// TwinCAT 3 PLC project CNC_Base_program
// ProgramVersion: 3.1.4020.1
// libraries:
//   Tc2_CncHli, * (Beckhoff Automation GmbH)
//   Tc2_ControllerToolbox, * (Beckhoff Automation GmbH)
//   Tc2_Drive, * (Beckhoff Automation GmbH)
//   Tc2_NcDrive, * (Beckhoff Automation GmbH)
//   Tc2_NCI, * (Beckhoff Automation GmbH)
//   Tc2_PlcInterpolation, * (Beckhoff Automation GmbH)
//   Tc2_Standard, * (Beckhoff Automation GmbH)
//   Tc2_System, * (Beckhoff Automation GmbH)
//   Tc2_Utilities, * (Beckhoff Automation GmbH)
//   Tc3_Module, * (Beckhoff Automation GmbH)
// project tree:
//   DUTs/Cnc_Data_Types/HMI/ ST_HmiAxis.TcDUT, ST_HmiChannel.TcDUT, ST_HmiData.TcDUT
//   DUTs/Cnc_Data_Types/ ST_BlockSearch.TcDUT, ST_CncChannel.TcDUT, ST_CncSystem.TcDUT, ST_PosVector.TcDUT, ST_MachineMode.TcDUT, ST_ManualModeParam.TcDUT, ST_OpModes.TcDUT, ST_OpStates.TcDUT, ST_SyntaxCheck.TcDUT
//   DUTs/Cnc_Data_Types/ToolManagement/ ST_ToolData.TcDUT, ST_ToolLife.TcDUT, ST_ToolManagement.TcDUT
//   DUTs/Recipe/ RecipeHeader_Struct.TcDUT, RecipeList_Struct.TcDUT
//   DUTs/VE_VarData/ ST_VEVariableConfig.TcDUT
//   / GlobalTextList.TcGTLO, PlcTask.TcTTO, Visualization Manager.TcVMO (not stored)
//   GVLs/ Global_Manual.TcGVL, Global_Variables.TcGVL, GVL.TcGVL, IOs.TcGVL, Machining_Data.TcGVL
//   POUs/ CncAxisEnable.TcPOU, CncHFunctions.TcPOU, CncPlcManualFunctions.TcPOU, CncPlcMessages.TcPOU, CncVariables.TcPOU, CncMFunctions.TcPOU, CncRefPosOffs.TcPOU, CncPlcProgram.TcPOU, MAIN.TcPOU
//   POUs/CNC/F1_Init/ CncToolControl.TcPOU, HLI_Init.TcPOU, HLI_AxisSetControlToPlc.TcPOU, HLI_ChannelSetControlToPlc.TcPOU, HLI_UserInitialisation.TcPOU
//   POUs/CNC/F2_Operation Mode/ HLI_AxisManualMode.TcPOU, HLI_AxisReset.TcPOU, HLI_ChannelModeAuto.TcPOU, HLI_ChannelModeManual.TcPOU, HLI_ChannelModeMDI.TcPOU, HLI_ChannelModeReference.TcPOU, HLI_ChannelModeStandby.TcPOU, HLI_ChannelReset.TcPOU, MM_TEst.TcPOU, HLI_CncChannel.TcPOU
//   POUs/CNC/F3_Control/ HLI_ChannelGetActiveFeed.TcPOU, HLI_ChannelGetStatusInfo.TcPOU, HLI_ChannelResetRequest.TcPOU, HLI_ChannelSetBackwardMotion.TcPOU, HLI_ChannelSetFeedHold.TcPOU, HLI_ChannelSetHandWheelIncs.TcPOU, HLI_ChannelSetOptionalM01Stop.TcPOU, HLI_ChannelSetProgramBlockIgnore.TcPOU, HLI_ChannelSetReducedFeed.TcPOU, HLI_ChannelSetSingleBlock.TcPOU, HLI_ChannelSetSuspendAxisOutput.TcPOU, HLI_ChannelSetSyntaxCheck.TcPOU, HLI_ChannelGetError.TcPOU, HLI_ChannelGetMessage.TcPOU, HLI_ChannelGetMode.TcPOU, HLI_ChannelGetState.TcPOU, HLI_AxisSetFeedHold.TcPOU, HLI_AxisSetReferenceCam.TcPOU, HLI_AxisSetTrackingOperation.TcPOU, HLI_ChannelSetOverride.TcPOU
//   POUs/CNC/F4_MHT-Function/ HLI_ChannelResetMFunctions.TcPOU, HLI_DoChannelHFunction.TcPOU, HLI_DoChannelMFunction.TcPOU, HLI_DoChannelTFunction.TcPOU, HLI_QuitAxisMFunction.TcPOU, HLI_QuitChannelMHTFunction.TcPOU
//   POUs/CNC/F5_Variables/ LinkVEChannelStructure.TcPOU
//   POUs/CNC/F6 BlockSearch/ FB_BlockSearchRead.TcPOU, FB_BlockSearchWrite.TcPOU, HLI_ChannelBlockSearch.TcPOU
//   POUs/CNC/F9_Misc/ ADSLOG.TcPOU, ADSLOG2.TcPOU, MySystemTime.TcPOU
//   POUs/CNC/F9_Misc/HandWheel/ FB_HandWheelEnc.TcPOU, PRG_ManualModeG201.TcPOU
//   POUs/CNC/F9_Misc/Security/ CheckCNCAlive.TcPOU, SetPlcAlive.TcPOU
//   POUs/General/ DemoTest.TcPOU, DemoUpDown.TcPOU, Examples.TcPOU, FB_Flash.TcPOU, FB_AdsRead.TcPOU, FB_ReadPParamValue.TcPOU, DemoSine.TcPOU, WritePersistentData.TcPOU
//   POUs/HMI/ CncHmiData.TcPOU, DIntToString.TcPOU, FB_ReadChannelData.TcPOU, LRealToString.TcPOU, FB_ReadTechnoTFunc.TcPOU, FB_ReadTechnoMFunc.TcPOU, FB_ReadTechnoGFunc.TcPOU, FB_ReadWriteFileData.TcPOU, SetHMIVariables.TcPOU
//   POUs/Messages/ FB_SimpleEventLog.TcPOU, ShowMessages.TcPOU
//   POUs/Temperature Controller/ PCamara.TcPOU, PCamara_Out.TcPOU, PExt.TcPOU, PExt_Out.TcPOU, PTab.TcPOU, PTab_Out.TcPOU, TController_Enable.TcPOU
// real-time tasks:
//   TASK PlcTask: cycle T#10ms, priority 20, ADS port 350
//   TASK VISU_TASK: cycle T#200000us, priority 30, ADS port 351
// motion (NC):
//   TASK NC-Task 1 SAF: cycle T#2ms, priority 4, ADS port 501
//   TASK NC-Task 1 SVB: cycle T#10ms, priority 9, ADS port 511
// I/O:
//   DEVICE Device 3 (EtherCAT), AmsNetId 192.168.200.135.4.1
//     Term 1 (EK1100) [EK1100 EtherCAT Coupler (2A E-Bus)]
//       Term 2 (EL1008) [EL1008 8Ch. Dig. Input 24V, 3ms]
//       Term 3 (EL1008) [EL1008 8Ch. Dig. Input 24V, 3ms]
//       Term 4 (EL2008) [EL2008 8Ch. Dig. Output 24V, 0.5A]
//       Term 5 (EL2008) [EL2008 8Ch. Dig. Output 24V, 0.5A]
//       Term 6 (EL4024) [EL4024 4Ch. Ana. Output 4-20mA, 12bit]
//       Term 7 (EL3318) [EL3318 8Ch. Ana Input Thermocouple (TC)]
//       Term 8 (EL7037) [EL7037 1Ch. Stepper motor output stage (24V, 1.5A)] // Motor AS1020
//       Term 9 (EL7037) [EL7037 1Ch. Stepper motor output stage (24V, 1.5A)]
//       Term 10 (EL7037) [EL7037 1Ch. Stepper motor output stage (24V, 1.5A)]
//       Term 11 (EL7037) [EL7037 1Ch. Stepper motor output stage (24V, 1.5A)]
//       Term 12 (EL7037) [EL7037 1Ch. Stepper motor output stage (24V, 1.5A)]
//       Term 13 (EL7037) [EL7037 1Ch. Stepper motor output stage (24V, 1.5A)]
//       Term 14 (EL7037) [EL7037 1Ch. Stepper motor output stage (24V, 1.5A)]
//       Term 15 (EL2522) [EL2522 2Ch. Pulse Train Output]
//       Term 32 (EL7037) [EL7037 1Ch. Stepper motor output stage (24V, 1.5A)]
//       Term 16 (EL9011) [EL9011 End Terminal]
// variable links:
//   CNC/Axes/B <-> Device 3 (EtherCAT)/Term 1 (EK1100)/Term 10 (EL7037)
//     Inputs/Enc_Counter <-> ENC Status compact/Counter value
//     Inputs/Enc_Latch <-> ENC Status compact/Latch value
//     Inputs/Enc_Status @bit 4 <-> ENC Status compact/Status/Counter overflow
//     Inputs/Enc_Status @bit 3 <-> ENC Status compact/Status/Counter underflow
//     Inputs/Enc_Status @bit 7 <-> ENC Status compact/Status/Extrapolation stall
//     Inputs/Enc_Status <-> ENC Status compact/Status/Latch C valid
//     Inputs/Enc_Status @bit 1 <-> ENC Status compact/Status/Latch extern valid
//     Inputs/Enc_Status @bit 2 <-> ENC Status compact/Status/Set counter done
//     Inputs/Enc_Status2 @bit 4 <-> ENC Status compact/Status/Status of extern latch
//     Inputs/Enc_Status2 <-> ENC Status compact/Status/Status of input A
//     Inputs/Enc_Status2 @bit 1 <-> ENC Status compact/Status/Status of input B
//     Inputs/Enc_Status2 @bit 2 <-> ENC Status compact/Status/Status of input C
//     Inputs/Enc_Status2 @bit 5 <-> ENC Status compact/Status/Sync error
//     Inputs/Enc_Status2 @bit 7 <-> ENC Status compact/Status/TxPDO Toggle
//     Inputs/STM_Status @bit 11 <-> STM Status/Status/Digital input 1
//     Inputs/STM_Status @bit 12 <-> STM Status/Status/Digital input 2
//     Inputs/STM_Status @bit 3 <-> STM Status/Status/Error
//     Inputs/STM_Status @bit 7 <-> STM Status/Status/Motor stall
//     Inputs/STM_Status @bit 5 <-> STM Status/Status/Moving negative
//     Inputs/STM_Status @bit 4 <-> STM Status/Status/Moving positive
//     Inputs/STM_Status @bit 1 <-> STM Status/Status/Ready
//     Inputs/STM_Status <-> STM Status/Status/Ready to enable
//     Inputs/STM_Status @bit 13 <-> STM Status/Status/Sync error
//     Inputs/STM_Status @bit 6 <-> STM Status/Status/Torque reduced
//     Inputs/STM_Status @bit 15 <-> STM Status/Status/TxPDO Toggle
//     Inputs/STM_Status @bit 2 <-> STM Status/Status/Warning
//     Outputs/Drv_Data_Out <-> STM Velocity/Velocity
//     Outputs/Enc_Ctrl <-> ENC Control compact/Control/Enable latch C
//     Outputs/Enc_Ctrl @bit 3 <-> ENC Control compact/Control/Enable latch extern on negative edge
//     Outputs/Enc_Ctrl @bit 1 <-> ENC Control compact/Control/Enable latch extern on positive edge
//     Outputs/Enc_Ctrl @bit 2 <-> ENC Control compact/Control/Set counter
//     Outputs/STM_Ctrl <-> STM Control/Control/Enable
//     Outputs/STM_Ctrl @bit 2 <-> STM Control/Control/Reduce torque
//     Outputs/STM_Ctrl @bit 1 <-> STM Control/Control/Reset
//   CNC/Axes/C <-> Device 3 (EtherCAT)/Term 1 (EK1100)/Term 13 (EL7037)
//     Inputs/Enc_Counter <-> ENC Status compact/Counter value
//     Inputs/Enc_Latch <-> ENC Status compact/Latch value
//     Inputs/Enc_Status @bit 4 <-> ENC Status compact/Status/Counter overflow
//     Inputs/Enc_Status @bit 3 <-> ENC Status compact/Status/Counter underflow
//     Inputs/Enc_Status @bit 7 <-> ENC Status compact/Status/Extrapolation stall
//     Inputs/Enc_Status <-> ENC Status compact/Status/Latch C valid
//     Inputs/Enc_Status @bit 1 <-> ENC Status compact/Status/Latch extern valid
//     Inputs/Enc_Status @bit 2 <-> ENC Status compact/Status/Set counter done
//     Inputs/Enc_Status2 @bit 4 <-> ENC Status compact/Status/Status of extern latch
//     Inputs/Enc_Status2 <-> ENC Status compact/Status/Status of input A
//     Inputs/Enc_Status2 @bit 1 <-> ENC Status compact/Status/Status of input B
//     Inputs/Enc_Status2 @bit 2 <-> ENC Status compact/Status/Status of input C
//     Inputs/Enc_Status2 @bit 5 <-> ENC Status compact/Status/Sync error
//     Inputs/Enc_Status2 @bit 7 <-> ENC Status compact/Status/TxPDO Toggle
//     Inputs/STM_Status @bit 11 <-> STM Status/Status/Digital input 1
//     Inputs/STM_Status @bit 12 <-> STM Status/Status/Digital input 2
//     Inputs/STM_Status @bit 3 <-> STM Status/Status/Error
//     Inputs/STM_Status @bit 7 <-> STM Status/Status/Motor stall
//     Inputs/STM_Status @bit 5 <-> STM Status/Status/Moving negative
//     Inputs/STM_Status @bit 4 <-> STM Status/Status/Moving positive
//     Inputs/STM_Status @bit 1 <-> STM Status/Status/Ready
//     Inputs/STM_Status <-> STM Status/Status/Ready to enable
//     Inputs/STM_Status @bit 13 <-> STM Status/Status/Sync error
//     Inputs/STM_Status @bit 6 <-> STM Status/Status/Torque reduced
//     Inputs/STM_Status @bit 15 <-> STM Status/Status/TxPDO Toggle
//     Inputs/STM_Status @bit 2 <-> STM Status/Status/Warning
//     Outputs/Drv_Data_Out <-> STM Velocity/Velocity
//     Outputs/Enc_Ctrl <-> ENC Control compact/Control/Enable latch C
//     Outputs/Enc_Ctrl @bit 3 <-> ENC Control compact/Control/Enable latch extern on negative edge
//     Outputs/Enc_Ctrl @bit 1 <-> ENC Control compact/Control/Enable latch extern on positive edge
//     Outputs/Enc_Ctrl @bit 2 <-> ENC Control compact/Control/Set counter
//     Outputs/STM_Ctrl <-> STM Control/Control/Enable
//     Outputs/STM_Ctrl @bit 2 <-> STM Control/Control/Reduce torque
//     Outputs/STM_Ctrl @bit 1 <-> STM Control/Control/Reset
//   CNC/Axes/Extruder <-> Device 3 (EtherCAT)/Term 1 (EK1100)/Term 32 (EL7037)
//     Inputs/Enc_Counter <-> ENC Status compact/Counter value
//     Inputs/Enc_Latch <-> ENC Status compact/Latch value
//     Inputs/Enc_Status @bit 4 <-> ENC Status compact/Status/Counter overflow
//     Inputs/Enc_Status @bit 3 <-> ENC Status compact/Status/Counter underflow
//     Inputs/Enc_Status @bit 7 <-> ENC Status compact/Status/Extrapolation stall
//     Inputs/Enc_Status <-> ENC Status compact/Status/Latch C valid
//     Inputs/Enc_Status @bit 1 <-> ENC Status compact/Status/Latch extern valid
//     Inputs/Enc_Status @bit 2 <-> ENC Status compact/Status/Set counter done
//     Inputs/Enc_Status2 @bit 4 <-> ENC Status compact/Status/Status of extern latch
//     Inputs/Enc_Status2 <-> ENC Status compact/Status/Status of input A
//     Inputs/Enc_Status2 @bit 1 <-> ENC Status compact/Status/Status of input B
//     Inputs/Enc_Status2 @bit 2 <-> ENC Status compact/Status/Status of input C
//     Inputs/Enc_Status2 @bit 5 <-> ENC Status compact/Status/Sync error
//     Inputs/Enc_Status2 @bit 7 <-> ENC Status compact/Status/TxPDO Toggle
//     Inputs/STM_Status @bit 11 <-> STM Status/Status/Digital input 1
//     Inputs/STM_Status @bit 12 <-> STM Status/Status/Digital input 2
//     Inputs/STM_Status @bit 3 <-> STM Status/Status/Error
//     Inputs/STM_Status @bit 7 <-> STM Status/Status/Motor stall
//     Inputs/STM_Status @bit 5 <-> STM Status/Status/Moving negative
//     Inputs/STM_Status @bit 4 <-> STM Status/Status/Moving positive
//     Inputs/STM_Status @bit 1 <-> STM Status/Status/Ready
//     Inputs/STM_Status <-> STM Status/Status/Ready to enable
//     Inputs/STM_Status @bit 13 <-> STM Status/Status/Sync error
//     Inputs/STM_Status @bit 6 <-> STM Status/Status/Torque reduced
//     Inputs/STM_Status @bit 15 <-> STM Status/Status/TxPDO Toggle
//     Inputs/STM_Status @bit 2 <-> STM Status/Status/Warning
//     Outputs/Drv_Data_Out <-> STM Velocity/Velocity
//     Outputs/Enc_Ctrl <-> ENC Control compact/Control/Enable latch C
//     Outputs/Enc_Ctrl @bit 3 <-> ENC Control compact/Control/Enable latch extern on negative edge
//     Outputs/Enc_Ctrl @bit 1 <-> ENC Control compact/Control/Enable latch extern on positive edge
//     Outputs/Enc_Ctrl @bit 2 <-> ENC Control compact/Control/Set counter
//     Outputs/STM_Ctrl <-> STM Control/Control/Enable
//     Outputs/STM_Ctrl @bit 2 <-> STM Control/Control/Reduce torque
//     Outputs/STM_Ctrl @bit 1 <-> STM Control/Control/Reset
//   CNC/Axes/X1 <-> Device 3 (EtherCAT)/Term 1 (EK1100)/Term 8 (EL7037)
//     Inputs/Enc_Counter <-> ENC Status compact/Counter value
//     Inputs/Enc_Latch <-> ENC Status compact/Latch value
//     Inputs/Enc_Status @bit 4 <-> ENC Status compact/Status/Counter overflow
//     Inputs/Enc_Status @bit 3 <-> ENC Status compact/Status/Counter underflow
//     Inputs/Enc_Status @bit 7 <-> ENC Status compact/Status/Extrapolation stall
//     Inputs/Enc_Status <-> ENC Status compact/Status/Latch C valid
//     Inputs/Enc_Status @bit 1 <-> ENC Status compact/Status/Latch extern valid
//     Inputs/Enc_Status @bit 2 <-> ENC Status compact/Status/Set counter done
//     Inputs/Enc_Status2 @bit 4 <-> ENC Status compact/Status/Status of extern latch
//     Inputs/Enc_Status2 <-> ENC Status compact/Status/Status of input A
//     Inputs/Enc_Status2 @bit 1 <-> ENC Status compact/Status/Status of input B
//     Inputs/Enc_Status2 @bit 2 <-> ENC Status compact/Status/Status of input C
//     Inputs/Enc_Status2 @bit 5 <-> ENC Status compact/Status/Sync error
//     Inputs/Enc_Status2 @bit 7 <-> ENC Status compact/Status/TxPDO Toggle
//     Inputs/STM_Status @bit 11 <-> STM Status/Status/Digital input 1
//     Inputs/STM_Status @bit 12 <-> STM Status/Status/Digital input 2
//     Inputs/STM_Status @bit 3 <-> STM Status/Status/Error
//     Inputs/STM_Status @bit 7 <-> STM Status/Status/Motor stall
//     Inputs/STM_Status @bit 5 <-> STM Status/Status/Moving negative
//     Inputs/STM_Status @bit 4 <-> STM Status/Status/Moving positive
//     Inputs/STM_Status @bit 1 <-> STM Status/Status/Ready
//     Inputs/STM_Status <-> STM Status/Status/Ready to enable
//     Inputs/STM_Status @bit 13 <-> STM Status/Status/Sync error
//     Inputs/STM_Status @bit 6 <-> STM Status/Status/Torque reduced
//     Inputs/STM_Status @bit 15 <-> STM Status/Status/TxPDO Toggle
//     Inputs/STM_Status @bit 2 <-> STM Status/Status/Warning
//     Outputs/Drv_Data_Out <-> STM Velocity/Velocity
//     Outputs/Enc_Ctrl <-> ENC Control compact/Control/Enable latch C
//     Outputs/Enc_Ctrl @bit 3 <-> ENC Control compact/Control/Enable latch extern on negative edge
//     Outputs/Enc_Ctrl @bit 1 <-> ENC Control compact/Control/Enable latch extern on positive edge
//     Outputs/Enc_Ctrl @bit 2 <-> ENC Control compact/Control/Set counter
//     Outputs/STM_Ctrl <-> STM Control/Control/Enable
//     Outputs/STM_Ctrl @bit 2 <-> STM Control/Control/Reduce torque
//     Outputs/STM_Ctrl @bit 1 <-> STM Control/Control/Reset
//   CNC/Axes/X2 <-> Device 3 (EtherCAT)/Term 1 (EK1100)/Term 9 (EL7037)
//     Inputs/Enc_Counter <-> ENC Status compact/Counter value
//     Inputs/Enc_Latch <-> ENC Status compact/Latch value
//     Inputs/Enc_Status @bit 4 <-> ENC Status compact/Status/Counter overflow
//     Inputs/Enc_Status @bit 3 <-> ENC Status compact/Status/Counter underflow
//     Inputs/Enc_Status @bit 7 <-> ENC Status compact/Status/Extrapolation stall
//     Inputs/Enc_Status <-> ENC Status compact/Status/Latch C valid
//     Inputs/Enc_Status @bit 1 <-> ENC Status compact/Status/Latch extern valid
//     Inputs/Enc_Status @bit 2 <-> ENC Status compact/Status/Set counter done
//     Inputs/Enc_Status2 @bit 4 <-> ENC Status compact/Status/Status of extern latch
//     Inputs/Enc_Status2 <-> ENC Status compact/Status/Status of input A
//     Inputs/Enc_Status2 @bit 1 <-> ENC Status compact/Status/Status of input B
//     Inputs/Enc_Status2 @bit 2 <-> ENC Status compact/Status/Status of input C
//     Inputs/Enc_Status2 @bit 5 <-> ENC Status compact/Status/Sync error
//     Inputs/Enc_Status2 @bit 7 <-> ENC Status compact/Status/TxPDO Toggle
//     Inputs/STM_Status @bit 11 <-> STM Status/Status/Digital input 1
//     Inputs/STM_Status @bit 12 <-> STM Status/Status/Digital input 2
//     Inputs/STM_Status @bit 3 <-> STM Status/Status/Error
//     Inputs/STM_Status @bit 7 <-> STM Status/Status/Motor stall
//     Inputs/STM_Status @bit 5 <-> STM Status/Status/Moving negative
//     Inputs/STM_Status @bit 4 <-> STM Status/Status/Moving positive
//     Inputs/STM_Status @bit 1 <-> STM Status/Status/Ready
//     Inputs/STM_Status <-> STM Status/Status/Ready to enable
//     Inputs/STM_Status @bit 13 <-> STM Status/Status/Sync error
//     Inputs/STM_Status @bit 6 <-> STM Status/Status/Torque reduced
//     Inputs/STM_Status @bit 15 <-> STM Status/Status/TxPDO Toggle
//     Inputs/STM_Status @bit 2 <-> STM Status/Status/Warning
//     Outputs/Drv_Data_Out <-> STM Velocity/Velocity
//     Outputs/Enc_Ctrl <-> ENC Control compact/Control/Enable latch C
//     Outputs/Enc_Ctrl @bit 3 <-> ENC Control compact/Control/Enable latch extern on negative edge
//     Outputs/Enc_Ctrl @bit 1 <-> ENC Control compact/Control/Enable latch extern on positive edge
//     Outputs/Enc_Ctrl @bit 2 <-> ENC Control compact/Control/Set counter
//     Outputs/STM_Ctrl <-> STM Control/Control/Enable
//     Outputs/STM_Ctrl @bit 2 <-> STM Control/Control/Reduce torque
//     Outputs/STM_Ctrl @bit 1 <-> STM Control/Control/Reset
//   CNC/Axes/Y <-> Device 3 (EtherCAT)/Term 1 (EK1100)/Term 14 (EL7037)
//     Inputs/Enc_Counter <-> ENC Status compact/Counter value
//     Inputs/Enc_Latch <-> ENC Status compact/Latch value
//     Inputs/Enc_Status @bit 4 <-> ENC Status compact/Status/Counter overflow
//     Inputs/Enc_Status @bit 3 <-> ENC Status compact/Status/Counter underflow
//     Inputs/Enc_Status @bit 7 <-> ENC Status compact/Status/Extrapolation stall
//     Inputs/Enc_Status <-> ENC Status compact/Status/Latch C valid
//     Inputs/Enc_Status @bit 1 <-> ENC Status compact/Status/Latch extern valid
//     Inputs/Enc_Status @bit 2 <-> ENC Status compact/Status/Set counter done
//     Inputs/Enc_Status2 @bit 4 <-> ENC Status compact/Status/Status of extern latch
//     Inputs/Enc_Status2 <-> ENC Status compact/Status/Status of input A
//     Inputs/Enc_Status2 @bit 1 <-> ENC Status compact/Status/Status of input B
//     Inputs/Enc_Status2 @bit 2 <-> ENC Status compact/Status/Status of input C
//     Inputs/Enc_Status2 @bit 5 <-> ENC Status compact/Status/Sync error
//     Inputs/Enc_Status2 @bit 7 <-> ENC Status compact/Status/TxPDO Toggle
//     Inputs/STM_Status @bit 11 <-> STM Status/Status/Digital input 1
//     Inputs/STM_Status @bit 12 <-> STM Status/Status/Digital input 2
//     Inputs/STM_Status @bit 3 <-> STM Status/Status/Error
//     Inputs/STM_Status @bit 7 <-> STM Status/Status/Motor stall
//     Inputs/STM_Status @bit 5 <-> STM Status/Status/Moving negative
//     Inputs/STM_Status @bit 4 <-> STM Status/Status/Moving positive
//     Inputs/STM_Status @bit 1 <-> STM Status/Status/Ready
//     Inputs/STM_Status <-> STM Status/Status/Ready to enable
//     Inputs/STM_Status @bit 13 <-> STM Status/Status/Sync error
//     Inputs/STM_Status @bit 6 <-> STM Status/Status/Torque reduced
//     Inputs/STM_Status @bit 15 <-> STM Status/Status/TxPDO Toggle
//     Inputs/STM_Status @bit 2 <-> STM Status/Status/Warning
//     Outputs/Drv_Data_Out <-> STM Velocity/Velocity
//     Outputs/Enc_Ctrl <-> ENC Control compact/Control/Enable latch C
//     Outputs/Enc_Ctrl @bit 3 <-> ENC Control compact/Control/Enable latch extern on negative edge
//     Outputs/Enc_Ctrl @bit 1 <-> ENC Control compact/Control/Enable latch extern on positive edge
//     Outputs/Enc_Ctrl @bit 2 <-> ENC Control compact/Control/Set counter
//     Outputs/STM_Ctrl <-> STM Control/Control/Enable
//     Outputs/STM_Ctrl @bit 2 <-> STM Control/Control/Reduce torque
//     Outputs/STM_Ctrl @bit 1 <-> STM Control/Control/Reset
//   CNC/Axes/Z1 <-> Device 3 (EtherCAT)/Term 1 (EK1100)/Term 11 (EL7037)
//     Inputs/Enc_Counter <-> ENC Status compact/Counter value
//     Inputs/Enc_Latch <-> ENC Status compact/Latch value
//     Inputs/Enc_Status @bit 4 <-> ENC Status compact/Status/Counter overflow
//     Inputs/Enc_Status @bit 3 <-> ENC Status compact/Status/Counter underflow
//     Inputs/Enc_Status @bit 7 <-> ENC Status compact/Status/Extrapolation stall
//     Inputs/Enc_Status <-> ENC Status compact/Status/Latch C valid
//     Inputs/Enc_Status @bit 1 <-> ENC Status compact/Status/Latch extern valid
//     Inputs/Enc_Status @bit 2 <-> ENC Status compact/Status/Set counter done
//     Inputs/Enc_Status2 @bit 4 <-> ENC Status compact/Status/Status of extern latch
//     Inputs/Enc_Status2 <-> ENC Status compact/Status/Status of input A
//     Inputs/Enc_Status2 @bit 1 <-> ENC Status compact/Status/Status of input B
//     Inputs/Enc_Status2 @bit 2 <-> ENC Status compact/Status/Status of input C
//     Inputs/Enc_Status2 @bit 5 <-> ENC Status compact/Status/Sync error
//     Inputs/Enc_Status2 @bit 7 <-> ENC Status compact/Status/TxPDO Toggle
//     Inputs/STM_Status @bit 11 <-> STM Status/Status/Digital input 1
//     Inputs/STM_Status @bit 12 <-> STM Status/Status/Digital input 2
//     Inputs/STM_Status @bit 3 <-> STM Status/Status/Error
//     Inputs/STM_Status @bit 7 <-> STM Status/Status/Motor stall
//     Inputs/STM_Status @bit 5 <-> STM Status/Status/Moving negative
//     Inputs/STM_Status @bit 4 <-> STM Status/Status/Moving positive
//     Inputs/STM_Status @bit 1 <-> STM Status/Status/Ready
//     Inputs/STM_Status <-> STM Status/Status/Ready to enable
//     Inputs/STM_Status @bit 13 <-> STM Status/Status/Sync error
//     Inputs/STM_Status @bit 6 <-> STM Status/Status/Torque reduced
//     Inputs/STM_Status @bit 15 <-> STM Status/Status/TxPDO Toggle
//     Inputs/STM_Status @bit 2 <-> STM Status/Status/Warning
//     Outputs/Drv_Data_Out <-> STM Velocity/Velocity
//     Outputs/Enc_Ctrl <-> ENC Control compact/Control/Enable latch C
//     Outputs/Enc_Ctrl @bit 3 <-> ENC Control compact/Control/Enable latch extern on negative edge
//     Outputs/Enc_Ctrl @bit 1 <-> ENC Control compact/Control/Enable latch extern on positive edge
//     Outputs/Enc_Ctrl @bit 2 <-> ENC Control compact/Control/Set counter
//     Outputs/STM_Ctrl <-> STM Control/Control/Enable
//     Outputs/STM_Ctrl @bit 2 <-> STM Control/Control/Reduce torque
//     Outputs/STM_Ctrl @bit 1 <-> STM Control/Control/Reset
//   CNC/Axes/Z2 <-> Device 3 (EtherCAT)/Term 1 (EK1100)/Term 12 (EL7037)
//     Inputs/Enc_Counter <-> ENC Status compact/Counter value
//     Inputs/Enc_Latch <-> ENC Status compact/Latch value
//     Inputs/Enc_Status @bit 4 <-> ENC Status compact/Status/Counter overflow
//     Inputs/Enc_Status @bit 3 <-> ENC Status compact/Status/Counter underflow
//     Inputs/Enc_Status @bit 7 <-> ENC Status compact/Status/Extrapolation stall
//     Inputs/Enc_Status <-> ENC Status compact/Status/Latch C valid
//     Inputs/Enc_Status @bit 1 <-> ENC Status compact/Status/Latch extern valid
//     Inputs/Enc_Status @bit 2 <-> ENC Status compact/Status/Set counter done
//     Inputs/Enc_Status2 @bit 4 <-> ENC Status compact/Status/Status of extern latch
//     Inputs/Enc_Status2 <-> ENC Status compact/Status/Status of input A
//     Inputs/Enc_Status2 @bit 1 <-> ENC Status compact/Status/Status of input B
//     Inputs/Enc_Status2 @bit 2 <-> ENC Status compact/Status/Status of input C
//     Inputs/Enc_Status2 @bit 5 <-> ENC Status compact/Status/Sync error
//     Inputs/Enc_Status2 @bit 7 <-> ENC Status compact/Status/TxPDO Toggle
//     Inputs/STM_Status @bit 11 <-> STM Status/Status/Digital input 1
//     Inputs/STM_Status @bit 12 <-> STM Status/Status/Digital input 2
//     Inputs/STM_Status @bit 3 <-> STM Status/Status/Error
//     Inputs/STM_Status @bit 7 <-> STM Status/Status/Motor stall
//     Inputs/STM_Status @bit 5 <-> STM Status/Status/Moving negative
//     Inputs/STM_Status @bit 4 <-> STM Status/Status/Moving positive
//     Inputs/STM_Status @bit 1 <-> STM Status/Status/Ready
//     Inputs/STM_Status <-> STM Status/Status/Ready to enable
//     Inputs/STM_Status @bit 13 <-> STM Status/Status/Sync error
//     Inputs/STM_Status @bit 6 <-> STM Status/Status/Torque reduced
//     Inputs/STM_Status @bit 15 <-> STM Status/Status/TxPDO Toggle
//     Inputs/STM_Status @bit 2 <-> STM Status/Status/Warning
//     Outputs/Drv_Data_Out <-> STM Velocity/Velocity
//     Outputs/Enc_Ctrl <-> ENC Control compact/Control/Enable latch C
//     Outputs/Enc_Ctrl @bit 3 <-> ENC Control compact/Control/Enable latch extern on negative edge
//     Outputs/Enc_Ctrl @bit 1 <-> ENC Control compact/Control/Enable latch extern on positive edge
//     Outputs/Enc_Ctrl @bit 2 <-> ENC Control compact/Control/Set counter
//     Outputs/STM_Ctrl <-> STM Control/Control/Enable
//     Outputs/STM_Ctrl @bit 2 <-> STM Control/Control/Reduce torque
//     Outputs/STM_Ctrl @bit 1 <-> STM Control/Control/Reset
//   TC3_IEC_CNC_Sample/TC3_IEC_CNC_Sample Instance <-> Device 3 (EtherCAT)/Term 1 (EK1100)/Term 2 (EL1008)
//     PlcTask Inputs/IOs.IO_In_B <-> Channel 3/Input
//     PlcTask Inputs/IOs.IO_In_Capaci <-> Channel 7/Input
//     PlcTask Inputs/IOs.IO_In_X1 <-> Channel 1/Input
//     PlcTask Inputs/IOs.IO_In_X2 <-> Channel 2/Input
//     PlcTask Inputs/IOs.IO_In_Y <-> Channel 6/Input
//     PlcTask Inputs/IOs.IO_In_Z1 <-> Channel 4/Input
//     PlcTask Inputs/IOs.IO_In_Z2 <-> Channel 5/Input
//   TC3_IEC_CNC_Sample/TC3_IEC_CNC_Sample Instance <-> Device 3 (EtherCAT)/Term 1 (EK1100)/Term 3 (EL1008)
//     PlcTask Inputs/IOs.IO_In_Emergencia <-> Channel 8/Input
//   TC3_IEC_CNC_Sample/TC3_IEC_CNC_Sample Instance <-> Device 3 (EtherCAT)/Term 1 (EK1100)/Term 4 (EL2008)
//     PlcTask Outputs/IOs.IO_Out_Aque_Extrusor <-> Channel 7/Output
//     PlcTask Outputs/IOs.IO_Out_Aque_Mesa <-> Channel 8/Output
//     PlcTask Outputs/IOs.IO_Out_HMI <-> Channel 4/Output
//     PlcTask Outputs/IOs.IO_Out_Vent_Camara <-> Channel 6/Output
//     PlcTask Outputs/IOs.IO_Out_Vent_Porta <-> Channel 5/Output
//     PlcTask Outputs/IOs.IO_Out_Vent_Quadro1 <-> Channel 2/Output
//     PlcTask Outputs/IOs.IO_Out_Vent_Quadro2 <-> Channel 3/Output
//     PlcTask Outputs/IOs.IO_Out_Vent_cabl_X <-> Channel 1/Output
//   TC3_IEC_CNC_Sample/TC3_IEC_CNC_Sample Instance <-> Device 3 (EtherCAT)/Term 1 (EK1100)/Term 5 (EL2008)
//     PlcTask Outputs/IOs.IO_Out_Chiller <-> Channel 1/Output
//   TC3_IEC_CNC_Sample/TC3_IEC_CNC_Sample Instance <-> Device 3 (EtherCAT)/Term 1 (EK1100)/Term 6 (EL4024)
//     PlcTask Outputs/IOs.A_Out_Aque_Ar <-> AO Outputs Channel 1/Analog output
//   TC3_IEC_CNC_Sample/TC3_IEC_CNC_Sample Instance <-> Device 3 (EtherCAT)/Term 1 (EK1100)/Term 7 (EL3318)
//     PlcTask Inputs/IOs.Temp_8 <-> TC Channel 8/Value
//     PlcTask Inputs/IOs.Temp_8_status[1] <-> TC Channel 8/Status/Underrange
//     PlcTask Inputs/IOs.Temp_8_status[2] <-> TC Channel 8/Status/Overrange
//     PlcTask Inputs/IOs.Temp_8_status[3] <-> TC Channel 8/Status/Error
//     PlcTask Inputs/IOs.Temp_8_status[4] <-> TC Channel 8/Status/TxPDO State
//     PlcTask Inputs/IOs.Temp_8_status[5] <-> TC Channel 8/Status/TxPDO Toggle
//     PlcTask Inputs/IOs.Temp_Cabos <-> TC Channel 7/Value
//     PlcTask Inputs/IOs.Temp_Cabos_status[1] <-> TC Channel 7/Status/Underrange
//     PlcTask Inputs/IOs.Temp_Cabos_status[2] <-> TC Channel 7/Status/Overrange
//     PlcTask Inputs/IOs.Temp_Cabos_status[3] <-> TC Channel 7/Status/Error
//     PlcTask Inputs/IOs.Temp_Cabos_status[4] <-> TC Channel 7/Status/TxPDO State
//     PlcTask Inputs/IOs.Temp_Cabos_status[5] <-> TC Channel 7/Status/TxPDO Toggle
//     PlcTask Inputs/IOs.Temp_Camara_in <-> TC Channel 1/Value
//     PlcTask Inputs/IOs.Temp_Camara_in_status[1] <-> TC Channel 1/Status/Underrange
//     PlcTask Inputs/IOs.Temp_Camara_in_status[2] <-> TC Channel 1/Status/Overrange
//     PlcTask Inputs/IOs.Temp_Camara_in_status[3] <-> TC Channel 1/Status/Error
//     PlcTask Inputs/IOs.Temp_Camara_in_status[4] <-> TC Channel 1/Status/TxPDO State
//     PlcTask Inputs/IOs.Temp_Camara_in_status[5] <-> TC Channel 1/Status/TxPDO Toggle
//     PlcTask Inputs/IOs.Temp_Camara_out <-> TC Channel 2/Value
//     PlcTask Inputs/IOs.Temp_Camara_out_status[1] <-> TC Channel 2/Status/Underrange
//     PlcTask Inputs/IOs.Temp_Camara_out_status[2] <-> TC Channel 2/Status/Overrange
//     PlcTask Inputs/IOs.Temp_Camara_out_status[3] <-> TC Channel 2/Status/Error
//     PlcTask Inputs/IOs.Temp_Camara_out_status[4] <-> TC Channel 2/Status/TxPDO State
//     PlcTask Inputs/IOs.Temp_Camara_out_status[5] <-> TC Channel 2/Status/TxPDO Toggle
//     PlcTask Inputs/IOs.Temp_Chiller <-> TC Channel 5/Value
//     PlcTask Inputs/IOs.Temp_Chiller_status[1] <-> TC Channel 5/Status/Underrange
//     PlcTask Inputs/IOs.Temp_Chiller_status[2] <-> TC Channel 5/Status/Overrange
//     PlcTask Inputs/IOs.Temp_Chiller_status[3] <-> TC Channel 5/Status/Error
//     PlcTask Inputs/IOs.Temp_Chiller_status[4] <-> TC Channel 5/Status/TxPDO State
//     PlcTask Inputs/IOs.Temp_Chiller_status[5] <-> TC Channel 5/Status/TxPDO Toggle
//     PlcTask Inputs/IOs.Temp_Extrusor_1 <-> TC Channel 4/Value
//     PlcTask Inputs/IOs.Temp_Extrusor_1_status[1] <-> TC Channel 4/Status/Underrange
//     PlcTask Inputs/IOs.Temp_Extrusor_1_status[2] <-> TC Channel 4/Status/Overrange
//     PlcTask Inputs/IOs.Temp_Extrusor_1_status[3] <-> TC Channel 4/Status/Error
//     PlcTask Inputs/IOs.Temp_Extrusor_1_status[4] <-> TC Channel 4/Status/TxPDO State
//     PlcTask Inputs/IOs.Temp_Extrusor_1_status[5] <-> TC Channel 4/Status/TxPDO Toggle
//     PlcTask Inputs/IOs.Temp_Quadro <-> TC Channel 6/Value
//     PlcTask Inputs/IOs.Temp_Quadro_status[1] <-> TC Channel 6/Status/Underrange
//     PlcTask Inputs/IOs.Temp_Quadro_status[2] <-> TC Channel 6/Status/Overrange
//     PlcTask Inputs/IOs.Temp_Quadro_status[3] <-> TC Channel 6/Status/Error
//     PlcTask Inputs/IOs.Temp_Quadro_status[4] <-> TC Channel 6/Status/TxPDO State
//     PlcTask Inputs/IOs.Temp_Quadro_status[5] <-> TC Channel 6/Status/TxPDO Toggle
//     PlcTask Inputs/IOs.Temp_Tabuleiro <-> TC Channel 3/Value
//     PlcTask Inputs/IOs.Temp_Tabuleiro_status[1] <-> TC Channel 3/Status/Underrange
//     PlcTask Inputs/IOs.Temp_Tabuleiro_status[2] <-> TC Channel 3/Status/Overrange
//     PlcTask Inputs/IOs.Temp_Tabuleiro_status[3] <-> TC Channel 3/Status/Error
//     PlcTask Inputs/IOs.Temp_Tabuleiro_status[4] <-> TC Channel 3/Status/TxPDO State
//     PlcTask Inputs/IOs.Temp_Tabuleiro_status[5] <-> TC Channel 3/Status/TxPDO Toggle

CONFIGURATION CNC_Base_program
    RESOURCE PLC ON TwinCAT3
        TASK PlcTask(INTERVAL := T#10ms, PRIORITY := 20);
        PROGRAM MAIN WITH PlcTask : MAIN;
    END_RESOURCE
END_CONFIGURATION

// ---- DUTs/Cnc_Data_Types/HMI/ST_HmiAxis.TcDUT
TYPE ST_HmiAxis :
STRUCT
	Name								: STRING;
	actCmdPosition					: LREAL;							(* mm *)
	actVelo							: LREAL;							(* mm/min *)
	actAcc							: LREAL;							(*  *)
	// ----------------------------
	current_position_acs			: LREAL;							(* mm *)
	active_position_acs			: LREAL;							(* mm *)
	end_position_acs				: LREAL;							(* mm *)
	distanceToGo					: LREAL;							(* mm *)
END_STRUCT
END_TYPE

// ---- DUTs/Cnc_Data_Types/HMI/ST_HmiChannel.TcDUT
TYPE ST_HmiChannel :
STRUCT
   SetModeAutomatic				: BOOL;
   SetModeManual					: BOOL;
   SetModeMDI						: BOOL;
	// ----------------------------
   SetStart							: BOOL;
   SetStop							: BOOL;
   SetReset							: BOOL;
	// ----------------------------
   State								: STRING;
   Mode								: STRING;
	CommandFeed						: LREAL;
	ActiveFeed						: LREAL;
	OverrideFeedrate				: LREAL;
	NcFileName						: STRING(255);
	NcFileOffset					: DINT;
	// ----------------------------
   Error								: BOOL;
   ErrorVis							: STRING;
	ActiveProgramBuffer			: ARRAY[0..2000] OF BYTE;
	// ----------------------------
	ActiveGFuncString				: STRING;
	ActiveMFuncString				: STRING;
	ActiveTFuncString				: STRING;
	// ----------------------------
	AxisMax							: INT;
	Axis								: ARRAY[0..5] OF ST_HmiAxis;
END_STRUCT
END_TYPE

// ---- DUTs/Cnc_Data_Types/HMI/ST_HmiData.TcDUT
TYPE ST_HmiData :
STRUCT
	NumberOfChannels				: UDINT;
	Channel							: ARRAY[0..5] OF ST_HmiChannel;
END_STRUCT
END_TYPE

// ---- DUTs/Cnc_Data_Types/ST_BlockSearch.TcDUT
TYPE ST_BlockSearch :
STRUCT
   (* Block Search *)
	Active         : BOOL;
   bStartRead     : BOOL;        (* Edge signal *)
   bStartWrite    : BOOL;        (* Edge signal *)
   nType          : INT;         (* 0 - no block search
                                    3 - start position by block count
                                    4 - start position by block nr
                                    5 - start position BY individual mark *)
   fDistance      : LREAL;
   bAutoReturn    : BOOL;
   nDeviationMax  : UDINT;
   nBlockNumber   : DINT;
   nPass          : DINT;
   nBlockCount    : DINT;
END_STRUCT
END_TYPE

// ---- DUTs/Cnc_Data_Types/ST_CncChannel.TcDUT
TYPE ST_CncChannel :
STRUCT
	Mode					: ST_OpModes;									(* Operation Mode *)
	State					: ST_OpStates;									(* Operation States *)

	ActMode				: UDINT;											(* Selected Mode *)
	ActModeString		: STRING;										(* Selected Mode as string *)
	ActState				: UDINT;											(* Selected State *)
	ActStateString		: STRING;										(* Selected State as string *)

	ActDistance			: LREAL;											(* Block Search : Act. Distance *)
	ActBlockCount  	: DINT;											(* Block Search : Act. Block Count *)

	M						: ARRAY [0..MAX_M_FUNCTIONS] OF BOOL;	(* M-Functions *)
	
	
	_M						: ARRAY [0..MAX_M_FUNCTIONS] OF BOOL;	(* only internal, quit M-Functions *)
	M_Argument			: ARRAY [0..MAX_M_FUNCTIONS] OF DINT;	(* Additional M-Function parameter *)

	H						: ARRAY [1..MAX_M_FUNCTIONS] OF BOOL;	(* H-Functions *)
	_H						: ARRAY [1..MAX_M_FUNCTIONS] OF BOOL;	(* only internal, quit H-Functions *)
	H_Argument			: ARRAY [1..MAX_M_FUNCTIONS] OF DINT;	(* Additional H-Function parameter *)

	T						: ARRAY [1..MAX_T_FUNCTIONS] OF BOOL;	(* T-Functions *)
	
	ProcessStartTime	: DT;												(* Process start time *)
	ProcessEndTime		: DT;												(* Process end time *)
	ProcessRunning		: BOOL;											(* Indicates that the process is running *)
	Error					: BOOL;											(* Fehlerflag des Kanals *)
	ErrorId				: UDINT;											(* FehlerId des Kanals *)
	ErrorMask			: HLI_ERROR_MASKE;							(* Informs the user about the error location in the cnc file *)

	Message				: STRING(HLI_MSG_CONTENT_STRL);			(* Message from NC program to PLC *)
END_STRUCT
END_TYPE

// ---- DUTs/Cnc_Data_Types/ST_CncSystem.TcDUT
TYPE ST_CncSystem :
STRUCT
	bHLIInit			: BOOL;		(* Initialization of HLI done *)
	bUserInitDone	: BOOL;		(* Initialization of user data done *)
	bInitError		: BOOL;		(* Error init HLI-Interfaces *)
	nInitErrorId	: UDINT;		(* ErrorId during init HLI-Interfaces *)
	Channel			: ARRAY[0..HLI_SYS_CH_MAX] OF ST_CncChannel;
	Tool				: ARRAY[0..MAX_TOOLS] OF CNC_TOOL_DATA; (* for external tool configuration, see SysMan. channel, SDA Param, Externe Werkzeugverwaltung *)
END_STRUCT
END_TYPE

// ---- DUTs/Cnc_Data_Types/ST_PosVector.TcDUT
TYPE ST_PosVector :
STRUCT
	fPosX				: LREAL;
	fPosY				: LREAL;
	fPosZ				: LREAL;
END_STRUCT
END_TYPE

// ---- DUTs/Cnc_Data_Types/ST_MachineMode.TcDUT
TYPE ST_MachineMode :
STRUCT
	(*Mode				: ST_OpModes;	*)	(* Operation Mode *)
	(*State				: ST_OpStates;*)	(* Operation States *)

	(* Operation Mode *)
	Standby			: BOOL;
	Manual			: BOOL;
	MDI				: BOOL;
	Automatic		: BOOL;
	Homing			: BOOL;

	(* Operation State *)
	Start				: BOOL;
	Stop				: BOOL;
	Reset				: BOOL;
	Error				: BOOL;

	(* Special functions *)
	DoSingleBlock	: BOOL;
	SingleBlock		: BOOL;
   FeedHold			: BOOL;
	Backward			: BOOL;
	PrgBlockIgnore	: BOOL;
	M01Stop			: BOOL;
	BlockSearch		: ST_BlockSearch;
	SyntaxCheck    : ST_SyntaxCheck;

	(* Strings *)
	ProgramName		: STRING(1024);
	MDIString		: STRING(1024);
END_STRUCT
END_TYPE

// ---- DUTs/Cnc_Data_Types/ST_ManualModeParam.TcDUT
TYPE ST_ManualModeParam :
STRUCT
	(* manual mode parameter *)
	nOpMode				: UINT;			(* operation mode, 0-no, 1-handwheel, 2-tip, 3-jog *)
	nLogAxisNr			: UINT;			(* number of the logical axis *)
	nControlElement	: UINT;			(* number of the logical control element *)
	nHandwheelNr		: UINT;			(* number of handwheel 1..max)*)
	nHandwheelIncs		: DINT;			(* number of handwheel increments *)
	nHandwheelRes		: DINT;			(* resolution of the handwheel*)
	nTipSpeed			: UDINT;			(* speed tip mode *)
	nJogSpeed			: UDINT;			(* speed jog mode *)
	nJogDistance		: UDINT;			(* jog distance *)
	bKeyPos				: BOOL;			(* key press positive *)
	bKeyNeg				: BOOL;			(* key press negative *)
	bKeyRapid			: BOOL;			(* key press rapid *)
END_STRUCT
END_TYPE

// ---- DUTs/Cnc_Data_Types/ST_OpModes.TcDUT
TYPE ST_OpModes :
STRUCT
	Standby			: BOOL;
	Auto				: BOOL;
	Manual			: BOOL;
	MDI				: BOOL;
	Homing			: BOOL;
END_STRUCT
END_TYPE

// ---- DUTs/Cnc_Data_Types/ST_OpStates.TcDUT
TYPE ST_OpStates :
STRUCT
	Selected			: BOOL;
	Ready				: BOOL;
	Start				: BOOL;
	Stop				: BOOL;
	Reset				: BOOL;
END_STRUCT
END_TYPE

// ---- DUTs/Cnc_Data_Types/ST_SyntaxCheck.TcDUT
TYPE ST_SyntaxCheck :
STRUCT
   (* SyntaxCheck *)
   nType          : INT;	(* 
										0x0000 ISG_STANDARD Normal mode
										0x0001 SV Block search
										0x0002 SOLLKON Offline Simulation with output of setpoint data
										0x0802 SOLLKON Offline Simulation without output of setpoint data
										0x0004 ON_LINE Simulation online visualisation
										0x0008 SYNCHK Simulation syntax check
										0x0010 PROD_TIME Simulation production time computation
										0x0020 ONLINE_PROD_TIME Simulation online production time computation
										0x0040 MACHINE_LOCK Dry run without axis movement
										0x0080 TECHNO_FILTER Dry run TECHNO filter
										0x0100 KIN_TRAFO_OFF Overwrites automatic enabling for kinematic transformations by a characteristic parameter defined in SDA_MDS (sda_mds*.lis).
									*)

END_STRUCT
END_TYPE

// ---- DUTs/Cnc_Data_Types/ToolManagement/ST_ToolData.TcDUT
TYPE ST_ToolData :		(* Tool data for a tool *)
STRUCT
(* -----------------------------------------
	Hint:
--------------------------------------------
	Do not modify
		- size or type of this struct

	only modify
		- name and comment of the tool parameters
-------------------------------------------- *)

		Nr							: INT;				(* Number of the tool *)
		ToolType					: INT;				(* Type of the tool *)
		SisterTool				: INT;				(* Sister tool number *)
		ToolLocked				: INT;				(* Tool locked = 1, else = 0 *)
		ParamInt1				: INT;				(* Free int parameter of the tool *)
		ParamInt2				: INT;				(* Free int parameter of the tool *)
		ParamInt3				: INT;				(* Free int parameter of the tool *)
		ParamInt4				: INT;				(* Free int parameter of the tool *)

		Length					: LREAL;				(* Length of the tool *)
		Radius					: LREAL;				(* Radius of the tool *)
		DeltaLength				: LREAL;				(* Oversize length of the tool *)
		DeltaRadius				: LREAL;				(* Oversize radius of the tool *)
		ToolLifeTime			: LREAL;				(* Tool Life Time *)
		ToolLifeTimeMax		: LREAL;				(* Tool Life Time Max *)
		ToolLifeDistance		: LREAL;				(* Tool Life Distance *)
		ToolLifeDistanceMax	: LREAL;				(* Tool Life Distance Max *)
		Param1					: LREAL;				(* Free parameter of the tool *)
		Param2					: LREAL;				(* Free parameter of the tool *)
		Param3					: LREAL;				(* Free parameter of the tool *)
		Param4					: LREAL;				(* Free parameter of the tool *)
		Param5					: LREAL;				(* Free parameter of the tool *)
		Param6					: LREAL;				(* Free parameter of the tool *)
		Param7					: LREAL;				(* Free parameter of the tool *)
		Param8					: LREAL;				(* Free parameter of the tool *)
		Param9					: LREAL;				(* Free parameter of the tool *)
		Param10					: LREAL;				(* Free parameter of the tool *)
		Param11					: LREAL;				(* Free parameter of the tool *)
		Param12					: LREAL;				(* Free parameter of the tool *)
		Param13					: LREAL;				(* Free parameter of the tool *)
		Param14					: LREAL;				(* Free parameter of the tool *)
		Param15					: LREAL;				(* Free parameter of the tool *)
		Param16					: LREAL;				(* Free parameter of the tool *)
		Param17					: LREAL;				(* Free parameter of the tool *)
		Param18					: LREAL;				(* Free parameter of the tool *)
		Param19					: LREAL;				(* Free parameter of the tool *)
		Param20					: LREAL;				(* Free parameter of the tool *)
		Param21					: LREAL;				(* Free parameter of the tool *)
		Param22					: LREAL;				(* Free parameter of the tool *)
		Param23					: LREAL;				(* Free parameter of the tool *)
		Param24					: LREAL;				(* Free parameter of the tool *)
		Param25					: LREAL;				(* Free parameter of the tool *)
		Param26					: LREAL;				(* Free parameter of the tool *)
		Param27					: LREAL;				(* Free parameter of the tool *)
		Param28					: LREAL;				(* Free parameter of the tool *)
		Param29					: LREAL;				(* Free parameter of the tool *)
		Param30					: LREAL;				(* Free parameter of the tool *)
		(*Name					: STRING;*)
END_STRUCT
END_TYPE

// ---- DUTs/Cnc_Data_Types/ToolManagement/ST_ToolLife.TcDUT
TYPE ST_ToolLife :		(* Tool life data for a tool *)
STRUCT
	tool_id			: DINT;		(* Id of the tool *)
	res				: DINT;
	time_used		: LREAL;		(* Time of used tool in seconds *)
	dist_used		: LREAL;		(* Distance of used tool in mm *)
END_STRUCT
END_TYPE

// ---- DUTs/Cnc_Data_Types/ToolManagement/ST_ToolManagement.TcDUT
TYPE ST_ToolManagement :		(* Tool management *)
STRUCT
		ToolLife					: ST_ToolLife;		(* tool life data, PLC -> HMI *)
		ToolDataActive			: BOOL;				(* tool data activation, HMI -> PLC *)
		ToolData					: ARRAY[1..MAX_TOOLS] OF ST_ToolData;		(* tool data, HMI -> PLC *)
END_STRUCT
END_TYPE

// ---- DUTs/Recipe/RecipeHeader_Struct.TcDUT
{attribute 'pack_mode':='1'}
TYPE RecipeHeader_Struct :
STRUCT
   Name1        : STRING[40];
   Name2        : STRING[40];
   Reserve      : ARRAY[3..10] OF STRING[40];
   Values       : ARRAY[1..30] OF LREAL;
   List         : ARRAY[1..50] OF RecipeList_Struct;
END_STRUCT
END_TYPE

// ---- DUTs/Recipe/RecipeList_Struct.TcDUT
{attribute 'pack_mode':='1'}
TYPE RecipeList_Struct :
STRUCT
   ToolId       : LREAL;
   PosX         : LREAL;
   PosY         : LREAL;
   PosZ         : LREAL;
   Tool1        : LREAL;
   Tool2        : LREAL;
   Tool3        : LREAL;
   GlueTime     : LREAL;
   Velo         : LREAL;
   Reserve      : ARRAY[10..20] OF LREAL;
END_STRUCT
END_TYPE

// ---- DUTs/VE_VarData/ST_VEVariableConfig.TcDUT
TYPE ST_VEVariableConfig :
STRUCT
	VARIABLE_1		: POINTER TO ARRAY[0..3] OF DINT;
	VARIABLE_2		: POINTER TO DINT;
	VARIABLE_3		: POINTER TO BOOL;
	VARIABLE_4		: POINTER TO DINT;
	VARIABLE_5		: POINTER TO DINT;
END_STRUCT
END_TYPE

// ---- GVLs/Global_Manual.TcGVL
VAR_GLOBAL
	(***********************************
	 * Declaration for 
	 * Manual functions
	 ************************************)
	PortalInfo				: STRING;
	PortalOn					: ARRAY[1..20] OF BOOL;
	PortalOff				: ARRAY[1..20] OF BOOL;
	PortalStatus			: ARRAY[1..20] OF BYTE;

	PortalSetValueLeft	: ARRAY[1..20] OF STRING;
	PortalActValueLeft	: ARRAY[1..20] OF STRING;
	PortalSetValueRight	: ARRAY[1..20] OF STRING;
	PortalActValueRight	: ARRAY[1..20] OF STRING;

	SchweissenInfo			: STRING;
	SchweissenOn			: ARRAY[1..20] OF BOOL;
	SchweissenOff			: ARRAY[1..20] OF BOOL;
	SchweissenStatus		: ARRAY[1..20] OF BYTE;

	WerkzeugInfo			: STRING;
	WerkzeugOn				: ARRAY[1..20] OF BOOL;
	WerkzeugOff				: ARRAY[1..20] OF BOOL;
	WerkzeugStatus			: ARRAY[1..20] OF BYTE;
	

END_VAR

// ---- GVLs/Global_Variables.TcGVL
VAR_GLOBAL CONSTANT
	FIRST_MESSAGE						: INT := 1;
	LAST_MESSAGE						: INT := 50;
	
	AXIS_MANUAL_KEYUNIT_MAX			: INT := 0;		(* [0..HLI_KEY_MAXIDX(11)], 0=1 KeyUnit, 1=2 KeyUnit, ... *)	
END_VAR

VAR_GLOBAL
	CncSystem							: ST_CncSystem;
	Axis1CurrPosition: LREAL;
	Axis2CurrPosition: LREAL;
	Axis3CurrPosition: LREAL;
END_VAR

// MK check
VAR_GLOBAL
	(*--------------------------*)
	(*	Connection variables     *)
	(*--------------------------*)

	(* General signals, only for starting BDE *)
	PlcMachineMode						: ARRAY[0..5] OF ST_MachineMode;	(* HMI -> PLC *)
	PLCSelectedChannel				: INT;			(* HMI -> PLC *)

	PlcFeedOverride					: UINT;			(* HMI -> PLC *)
	PlcFeedOverride2					: UINT;			(* HMI -> PLC *)
	PlcSpindleOverride				: UINT;			(* HMI -> PLC *)

	(* PLC control signals *)
	PlcAxisEnable						: BOOL;			(* HMI -> PLC *)
	PlcDeleteFailure					: BOOL;			(* HMI -> PLC *)

	PlcReset								: BOOL;
	PlcVarWriteSettings				: BOOL;


	PlcArrayInt							: ARRAY[0..20] OF INT;
	PlcArrayReal						: ARRAY[0..10] OF REAL;
	PlcArrayString3					: ARRAY[0..10] OF STRING(50);
	PlcArrayString						: ARRAY[0..10] OF STRING;

	(* Function keys 5, 6 and 7 on the right side *)
	PlcFKeyRight5						: BOOL;
	PlcFKeyRight6						: BOOL;
	PlcFKeyRight7						: BOOL;
	
	(*--------------------------*)
	(*	BDE, PLC -> HMI          *)
	(*--------------------------*)
	BDEControlOn						: BOOL;
	BDEAutomatic						: BOOL;
	BDEVarBoolTimer					: ARRAY[0..10] OF BOOL;
	BDEVarBoolCounter					: ARRAY[0..10] OF BOOL;
	BDEVarBoolMessage					: ARRAY[0..50] OF BOOL;
	
	(* Manual Mode *)
	PlcManualModeLeftKey				: BOOL;
	PlcManualModeRightKey			: BOOL;
	PlcManualModeRapidFeedKey		: BOOL;
	PlcManualModeSelectedAxis		: UINT;
	PlcManualModeSpeed				: UDINT;
	PlcManualModeIncrements			: UDINT;
	PlcManualModeOpMode				: UINT;	(* 1-handwheel, 2-continuous, 3-Incremental, ... *)
	PlcManualModeHandWheelIncs		: DINT;
	PlcManualModeHandWheelRes		: DINT := 1;

	(*--------------------------*)
	(* Tool management          *)
	(*--------------------------*)
	PlcToolManagement					: ST_ToolManagement;
	
   (*--------------------------*)
   (* Recipe HMI -> PLC        *)
   (*--------------------------*)
   RecipeData							: RecipeHeader_Struct;
	
END_VAR

VAR_GLOBAL
	(*--------------------------*)
	(*	Messages                 *)
	(*--------------------------*)
	MSGList1								: ARRAY [FIRST_MESSAGE..LAST_MESSAGE] OF BOOL;
	MSGListQuit1						: ARRAY [FIRST_MESSAGE..LAST_MESSAGE] OF BOOL;
	MSGList2								: ARRAY [FIRST_MESSAGE..LAST_MESSAGE] OF BOOL;
	MSGListQuit2						: ARRAY [FIRST_MESSAGE..LAST_MESSAGE] OF BOOL;
	MSGList3								: ARRAY [FIRST_MESSAGE..LAST_MESSAGE] OF BOOL;
	MSGListQuit3						: ARRAY [FIRST_MESSAGE..LAST_MESSAGE] OF BOOL;
	MSGList4								: ARRAY [FIRST_MESSAGE..LAST_MESSAGE] OF BOOL;
	MSGListQuit4						: ARRAY [FIRST_MESSAGE..LAST_MESSAGE] OF BOOL;
END_VAR

VAR_GLOBAL PERSISTENT
	test1									: INT;
	test2									: INT;
	test3									: INT;
END_VAR

VAR_GLOBAL
	(*--------------------------*)
	(*	Temperatura             *)
	(*--------------------------*)
	Temp_Camara_set			: DINT :=0;						(*0.01ºC*)
	Temp_Tabuleiro_set		: DINT :=0;						(*0.01ºC*)
	Temp_Extrusor_1_set		: DINT :=0;						(*0.1ºC*)
	Temp_Extrusor_2_set		: DINT :=0;						(*0.1ºC*)

END_VAR

// ---- GVLs/GVL.TcGVL
{attribute 'qualified_only'}
VAR_GLOBAL
	Temp_Camara_in :INT;
	Temp_Tabuleiro :INT;
	Temp_Extrusor_1 :INT;
	Temp_Chiller :INT;
	Temp_Quadro :INT;
	Temp_Cabos:INT;
	Temp_8:INT;
	Temp_MotorB:LREAL:=50.0;
	Temp_PontoMovel:LREAL:=50.0;
	gvl_bstate_start :BOOL:= FALSE;
	gvl_sprogramname :STRING(500) := '';
	gvl_currentState :DWORD;
	gvl_automaticstop :BOOL :=FALSE;
	gvl_automaticreset :BOOL :=FALSE;
	gvl_automaticselected :BOOL :=FALSE;
	gvl_bEnableTracking:BOOL:=FALSE;
	gvl_plcAxisEnable:BOOL:=FALSE;
	gvl_operationMode:STRING(100):='';
	gvl_manualMode:BOOL;
	gvl_automaticMode:BOOL;
	gvl_machine_state:STRING(500):='';
	gvl_blockcount:DINT:=0;
	gvl_aquecimento_mesa:BOOL :=FALSE;
	gvl_aquecimento_extrusor:BOOL :=FALSE;
	gvl_manualmode_isactivated:BOOL :=FALSE;
	gvl_manualmode_busy:BOOL :=FALSE;
	gvl_currentMode:DWORD;
	gvl_Manual_nOpMode:UINT;
END_VAR

// ---- GVLs/IOs.TcGVL
VAR_GLOBAL
	IO_In1				AT %I*		: BOOL;
	IO_In2				AT %I*		: BOOL;
	IO_In3				AT %I*		: BOOL;
	IO_In4				AT %I*		: BOOL;

	IO_Out1				AT %Q*		: BOOL;
	IO_Out2				AT %Q*		: BOOL;
	IO_Out3				AT %Q*		: BOOL;
	IO_Out4				AT %Q*		: BOOL;
	
	
	//Definição dos inputs/outputs cartas de I/O
	
	IO_Out_Vent_cabl_X	AT %Q*		: BOOL;
	IO_Out_Vent_Quadro1	AT %Q*		: BOOL;
	IO_Out_Vent_Quadro2	AT %Q*		: BOOL;
	IO_Out_HMI			AT %Q*		: BOOL;
	IO_Out_Vent_Porta	AT %Q*		: BOOL;
	IO_Out_Vent_Camara	AT %Q*		: BOOL;
	IO_Out_Aque_Extrusor	AT %Q*		: BOOL;
	IO_Out_Aque_Mesa	AT %Q*		: BOOL;
	IO_Out_Chiller		AT %Q*		: BOOL;
	A_Out_Aque_Ar		AT %Q*		: UINT;
	
	IO_In_X1			AT %I*		: BOOL;
	IO_In_X2			AT %I*		: BOOL;
	IO_In_B				AT %I*		: BOOL;
	IO_In_Z1			AT %I*		: BOOL;
	IO_In_Z2			AT %I*		: BOOL;
	IO_In_Y				AT %I*		: BOOL;
	IO_In_Capaci		AT %I*		: BOOL;
	IO_In_Emergencia	AT %I*		: BOOL;
	
	//Inputs Temperatura
	
	Temp_Camara_in			AT %I*			: INT;						(*0.01ºC*)
	Temp_Camara_in_status	AT %I*			: ARRAY [1..5] OF BOOL;		(*Underrange; Overrange; Error; TxPDO State; TxPDO Toggle*)
	
	Temp_Camara_out			AT %I*			: INT;						(*0.01ºC*)
	Temp_Camara_out_status	AT %I*			: ARRAY [1..5] OF BOOL;		(*Underrange; Overrange; Error; TxPDO State; TxPDO Toggle*)
	
	Temp_Tabuleiro			AT %I*			: INT;						(*0.01ºC*)
	Temp_Tabuleiro_status	AT %I*			: ARRAY [1..5] OF BOOL;		(*Underrange; Overrange; Error; TxPDO State; TxPDO Toggle*)
	
	Temp_Extrusor_1			AT %I*			: INT;						(*0.1ºC*)
	Temp_Extrusor_1_status	AT %I*			: ARRAY [1..5] OF BOOL;		(*Underrange; Overrange; Error; TxPDO State; TxPDO Toggle*)
	
	Temp_Chiller			AT %I*			: INT;						(*0.1ºC*)
	Temp_Chiller_status		AT %I*			: ARRAY [1..5] OF BOOL;		(*Underrange; Overrange; Error; TxPDO State; TxPDO Toggle*)
	
	Temp_Quadro				AT %I*			: INT;						(*0.1ºC*)
	Temp_Quadro_status		AT %I*			: ARRAY [1..5] OF BOOL;		(*Underrange; Overrange; Error; TxPDO State; TxPDO Toggle*)
	
	Temp_Cabos				AT %I*			: INT;						(*0.1ºC*)
	Temp_Cabos_status		AT %I*			: ARRAY [1..5] OF BOOL;		(*Underrange; Overrange; Error; TxPDO State; TxPDO Toggle*)
	
	Temp_8					AT %I*			: INT;						(*0.1ºC*)
	Temp_8_status			AT %I*			: ARRAY [1..5] OF BOOL;		(*Underrange; Overrange; Error; TxPDO State; TxPDO Toggle*)
	
END_VAR

// ---- GVLs/Machining_Data.TcGVL
VAR_GLOBAL CONSTANT
	(* General limits *)
	MAX_TOOLS								: UINT := 50;
	SystemToolNr							: INT := 30;		(* System Tool Number *)
	
	MAX_TIMER								: INT := 50;
	MAX_M_FUNCTIONS						: UDINT := 200;
	MAX_T_FUNCTIONS						: UDINT := 200;

	(* BDE - Messages *)
	BDE_MSG_1								: INT := 1;
	BDE_MSG_2								: INT := 2;
	BDE_MSG_3								: INT := 3;

	(* BDE - Timer *)
	BDE_TIMER_SUM							: INT := 1;
	BDE_TIMER_CONTROL_ON					: INT := 2;
	BDE_TIMER_AUTOMATIC					: INT := 3;
	BDE_TIMER_ERROR						: INT := 4;

	(* BDE - Counter *)
	BDE_COUNTER_AUTO						: INT := 1;
	BDE_COUNTER_PIECES					: INT := 2;
END_VAR

VAR_GLOBAL
	(*--------------------------*)
	(*	Machine data table       *)
	(*--------------------------*)
	PLCMParBool				: ARRAY[1..10] OF BOOL;
	PLCMParInt				: ARRAY[1..50] OF INT;
	PLCMParByte				: ARRAY[1..20] OF BYTE;
	PLCMParDInt				: ARRAY[1..70] OF DINT;
	PLCMParUSInt			: ARRAY[1..20] OF USINT;
	PLCMParUInt				: ARRAY[1..20] OF UINT;
	PLCMParUDInt			: ARRAY[1..20] OF UDINT;
	PLCMParReal				: ARRAY[1..90] OF REAL;
	PLCMParLReal			: ARRAY[1..90] OF LREAL;
	PLCMParString			: ARRAY[1..50] OF STRING;
	PLCMParTime				: ARRAY[1..50] OF TIME;

	PLCMParList1			: ARRAY[1..100] OF LREAL;
	PLCMParList2			: ARRAY[1..50] OF LREAL;
	PLCMParList3			: ARRAY[1..50] OF LREAL;
	PLCMParListString		: ARRAY[1..50] OF STRING;
	PLCMParTimer			: ARRAY[1..50] OF TIME;
END_VAR

VAR_GLOBAL
	(* Timer *)
	PlcTimer					: ARRAY[1..MAX_TIMER] OF REAL;

	(* General Machining data *)
	MachineParam			: ARRAY[1..50] OF REAL;
	TestBol					: ARRAY[1..50] OF BOOL;
END_VAR

// ---- POUs/MAIN.TcPOU
PROGRAM MAIN

(* ========================================================= *)
(*    PRG: TwinCAT CNC                                       *)
(* --------------------------------------------------------- *)
(*  Desc: Base PLC program for TwinCAT CNC                  *)
(* 	Author: MK                                                *)
(*  Date: 21.12.2011                                        *)
(*  Cust.:                                                   *)
(*  M-No:                                                   *)
(*  Kom.:                                                   *)
(*  Rev.: 1.3  from 1.24                                    *)
(* ========================================================= *)

DemoSine();
DemoUpDown();
DemoTest();
WritePersistentData();
ShowMessages();
MySystemTime();

HLI_Init();
IF CncSystem.bHLIInit = TRUE THEN
	CncPlcProgram();
	CncMFunctions();
	CncPlcManualFunctions();
	CncPlcMessages();
	CncRefPosOffs();
	CncVariables();
	CncHmiData();
	
	//gpAx[0]^.ipo_mc_control.emergency_stop.command_w :=1;
	
	//Axis1CurrPosition := gpAx[0]^.lr_state.current_position_acs_r/10000.0;
	//Axis2CurrPosition := gpAx[0]^.lr_state.current_position_acs_r/10000.0;
	//Axis3CurrPosition := gpAx[0]^.lr_state.current_position_acs_r/10000.0;
	
END_IF



								(*--Belo Controlador--*)
TController_Enable();
								
								(* -- Set das variáveis para a HMI -- *)
SetHMIVariables();

END_PROGRAM

// ---- POUs/General/DemoSine.TcPOU
PROGRAM DemoSine
VAR
	X_Value		: REAL;
	Y_Value		: REAL;
	Y_ValueAbs	: REAL;

	maxValue		: INT := 1000;
	index			: INT;
END_VAR

(* ========================================================= *)
(*    PRG: DemoSine                                          *)
(* --------------------------------------------------------- *)
(*   Desc: Example, shows how to generate a sine             *)
(* Author: MK                                                *)
(*   Date: 21.12.2011                                        *)
(*   Rev.: 1.0                                               *)
(* ========================================================= *)


IF index >= maxValue THEN
	index := 0;
ELSE
	index := index + 1;
END_IF

X_Value := INT_TO_REAL(index)/INT_TO_REAL(maxValue) * 2.0 * 3.1415;
Y_Value := SIN(X_Value) * 100.0;
Y_ValueAbs := (Y_Value+100.0)/2.0;

END_PROGRAM

// ---- POUs/General/DemoUpDown.TcPOU
PROGRAM DemoUpDown
VAR
	bGo				: BOOL;
	UpDown			: INT;
END_VAR

(* ========================================================= *)
(*    PRG: DemoUpDown                                        *)
(* --------------------------------------------------------- *)
(*   Desc: Example, shows how to generate a up down signal   *)
(* Author: MK                                                *)
(*   Date: 21.12.2011                                        *)
(*   Rev.: 1.0                                               *)
(* ========================================================= *)


(* up down counter *)
IF bGo THEN
	UpDown := UpDown - 1;
	IF UpDown < 1 THEN
		bGo := FALSE;
	END_IF
ELSE
	UpDown := UpDown + 1;
	IF UpDown >= 100 THEN
		bGo := TRUE;
	END_IF
END_IF

END_PROGRAM

// ---- POUs/General/DemoTest.TcPOU

PROGRAM DemoTest
VAR_INPUT
	bEnable					: BOOL := TRUE;
END_VAR
VAR
	HandWheelEnc			: FB_HandWheelEnc;
	incs						: UDINT;
	dir						: INT;
	testTOD					: TOD;
	testDT					: DT;
	testTime					: TIME;
	testUInt32				: UDINT;
	nColor					: UDINT := 16#5522AA;
	stPosVector				: ST_PosVector;
END_VAR

IF bEnable = TRUE THEN
	PortalActValueLeft[3] := INT_TO_STRING(DemoUpDown.UpDown);
	PortalActValueLeft[4] := INT_TO_STRING(DemoUpDown.UpDown);
	PortalActValueLeft[5] := INT_TO_STRING(DemoUpDown.UpDown);
END_IF


IF dir = 0 THEN
	;
ELSIF dir = 1 THEN
	incs := incs + 1;
	
	IF incs > 1024 THEN
		incs := 0;
	END_IF
ELSIF dir = 2 THEN 
	incs := incs - 1;

	IF incs < 0 THEN
		incs := 1024;
	END_IF
END_IF

HandWheelEnc(EncoderValue:=incs);


stPosVector.fPosX := CncHmiData.PlcHmiData.Channel[0].Axis[0].active_position_acs;
stPosVector.fPosY := CncHmiData.PlcHmiData.Channel[0].Axis[1].active_position_acs;
stPosVector.fPosZ := CncHmiData.PlcHmiData.Channel[0].Axis[2].active_position_acs;

END_PROGRAM

// ---- POUs/CNC/F9_Misc/HandWheel/FB_HandWheelEnc.TcPOU
FUNCTION_BLOCK FB_HandWheelEnc
VAR_INPUT
   EncoderValue         : UDINT;
   EncoderValueMax      : DINT := 65535;		//  := 1024;
END_VAR
VAR_OUTPUT
   OUT                  : DINT;
END_VAR
VAR
   oldEncoderValue      : UDINT;
   nTurns               : DINT;
END_VAR

(* ========================================================= *)
(*     FB: FB_HandWheelEnc                                   *)
(* --------------------------------------------------------- *)
(*   Desc: Handles encoder overflow                          *)
(* Author: MK                                                *)
(*   Date: 20.10.2015                                        *)
(*   Rev.: 1.1                                               *)
(* ========================================================= *)


IF UDINT_TO_DINT(oldEncoderValue - EncoderValue) >  EncoderValueMax/2 THEN		// positiv overflow
	nTurns := nTurns + 1;
ELSIF UDINT_TO_DINT(EncoderValue - oldEncoderValue) > EncoderValueMax/2 THEN	// negativ overflow
	nTurns := nTurns - 1;
END_IF

oldEncoderValue := EncoderValue;

OUT := nTurns * EncoderValueMax + UDINT_TO_DINT(EncoderValue);

END_FUNCTION_BLOCK

// ---- POUs/HMI/CncHmiData.TcPOU
PROGRAM CncHmiData
VAR_INPUT
END_VAR
VAR
	PlcHmiData						: ST_HmiData;
	nChIdx							: UDINT;
	fbReadChannelData				: ARRAY[0..5] OF FB_ReadChannelData;
END_VAR

(* ========================================================= *)
(*    FUN: CncHmiData                                        *)
(* --------------------------------------------------------- *)
(*   Desc:                                                   *)
(* Author: MK                                                *)
(*   Date: 01.12.2015                                        *)
(*   Rev.: 1.0                                               *)
(* ========================================================= *)


//RETURN;

PlcHmiData.NumberOfChannels := gpPform^.nc_config.number_of_channels_r;
FOR nChIdx := 0 TO PlcHmiData.NumberOfChannels - 1 DO
	fbReadChannelData[nChIdx](nChIdx:=nChIdx, pHmiChannel:=ADR(PlcHmiData.Channel[nChIdx]));
END_FOR

END_PROGRAM

// ---- POUs/HMI/FB_ReadChannelData.TcPOU
FUNCTION_BLOCK FB_ReadChannelData
VAR_INPUT
	nChIdx							: UDINT;
	pHmiChannel						: POINTER TO ST_HmiChannel;
END_VAR
VAR_OUTPUT
END_VAR
VAR
	pChannel							: POINTER TO HIGH_LEVEL_INTERFACE_CH;
	pAx								: POINTER TO HIGH_LEVEL_INTERFACE_AX;

	timerFileName					: TON;
	sFileName						: STRING(255);
	sFileNameOld					: STRING(255);
	sTmp								: STRING(255);

	nFileOffset						: DINT;
	nFileOffsetOld					: DINT := -1;
	
	fbReadWriteData				: FB_ReadWriteFileData;
	bReadFileErr					: BOOL;
	bReadNcFile						: BOOL;
	bReadFileActive				: BOOL;

	timerTechno						: TON;
	bReadTechnoInfoActive		: BOOL;	
	fbReadTechnoGFunc				: FB_ReadTechnoGFunc;
	fbReadTechnoMFunc				: FB_ReadTechnoMFunc;
	fbReadTechnoTFunc				: FB_ReadTechnoTFunc;
	
	fbFlash							: FB_Flash;
	nAxIdx							: INT;
END_VAR

(* ========================================================= *)
(*    FUN: FB_ReadChannelData                                *)
(* --------------------------------------------------------- *)
(*   Desc:                                                   *)
(* Author: MK                                                *)
(*   Date: 01.12.2015                                        *)
(*   Rev.: 1.0                                               *)
(* ========================================================= *)


(* get pointer to channel data *)
pChannel := gpCh[nChIdx];
IF pChannel = 0 THEN
	RETURN;
END_IF

(* commanded feedrade *)
pHmiChannel^.CommandFeed := pChannel^.bahn_state.command_feed_r/1000.0*60.0;		(* mm/min *)

(* active feedrade *)
pHmiChannel^.ActiveFeed := pChannel^.bahn_state.active_feed_r/1000.0*60.0;			(* mm/min *)

(* override *)
pHmiChannel^.OverrideFeedrate := pChannel^.bahn_mc_control.override_feedrate.state_r/10.0;		(* % *)


(* read file name and file offset *)
timerFileName(IN := NOT(timerFileName.Q), PT := T#150MS);
IF timerFileName.Q THEN
	(*MRODRIGUES
	sFileName := pChannel^.bahn_state.file_name_r.zeichen;*)
	sFileName := GVL.gvl_sprogramname;
	nFileOffset := pChannel^.bahn_state.active_fileoffset_r;
	pHmiChannel^.NcFileName := sFileName;
	pHmiChannel^.NcFileOffset := nFileOffset;

	IF sFileNameOld <> sFileName OR nFileOffsetOld <> nFileOffset THEN
		sFileNameOld := sFileName;
		nFileOffsetOld := nFileOffset;
		bReadNcFile := TRUE;
	END_IF
END_IF

(* read nc file data *)
IF (bReadNcFile = TRUE OR bReadFileActive = TRUE) THEN
	IF sFileName = ''  
		OR LEFT(STR:=sFileName, SIZE:=3) = 'C:\'
	THEN
		sTmp := sFileName;
	ELSE
		(* sub program, add default path *)
		sTmp := CONCAT('c:\twincat\cnc\', sFileName);
	END_IF
	
	fbReadWriteData(sNetId := '',
							sPathName := sTmp,
							nSeekPos := pHmiChannel^.NcFileOffset,
							bExecute := bReadNcFile,
							bWrite := FALSE,
							pBuffer := ADR(pHmiChannel^.ActiveProgramBuffer),
							nBufferSize := SIZEOF(pHmiChannel^.ActiveProgramBuffer)-1,
							bError => bReadFileErr,
							bBusy => bReadFileActive);
	bReadNcFile := FALSE;

	IF fbReadWriteData.bBusy = FALSE AND fbReadWriteData.bError = FALSE THEN
		bReadFileErr := FALSE;
	END_IF
END_IF


(* read technology information *)
timerTechno(IN := NOT(timerTechno.Q), PT := T#500MS);
IF timerTechno.Q THEN
	bReadTechnoInfoActive := TRUE;
END_IF

IF bReadTechnoInfoActive THEN
	fbReadTechnoGFunc(nIdxGrp	:= 16#20100 + 1 + nChIdx,
							nIdxOffs	:= 16#03C,
							nLen		:= 2*40,
							bStart	:= timerTechno.Q,
							pStr		:= ADR(pHmiChannel^.ActiveGFuncString));
							
	fbReadTechnoMFunc(nIdxGrp	:= 16#20100 + 1 + nChIdx,
							nIdxOffs	:= 16#03D,
							nLen		:= 4*40,
							bStart	:= timerTechno.Q,
							pStr		:= ADR(pHmiChannel^.ActiveMFuncString));

	fbReadTechnoTFunc(nIdxGrp	:= 16#20100 + 1 + nChIdx,
							nIdxOffs	:= 16#01A,
							nLen		:= 4,
							bStart	:= timerTechno.Q,
							pStr		:= ADR(pHmiChannel^.ActiveTFuncString));
							
	IF fbReadTechnoGFunc.bBusy = FALSE
		AND fbReadTechnoMFunc.bBusy = FALSE
		AND fbReadTechnoTFunc.bBusy = FALSE
	THEN
		bReadTechnoInfoActive := FALSE;
	END_IF
END_IF


(* channel mode and state *) 
pHmiChannel^.Mode := CncSystem.Channel[nChIdx+1].ActModeString;
pHmiChannel^.State := CncSystem.Channel[nChIdx+1].ActStateString;


(* channel mode Automatic, Manual, MDI *)
IF pHmiChannel^.SetModeAutomatic = TRUE THEN
	PlcMachineMode[nChIdx+1].Automatic := pHmiChannel^.SetModeAutomatic;
	pHmiChannel^.SetModeAutomatic := FALSE;
	IF PlcMachineMode[nChIdx+1].ProgramName = '' THEN
		PlcMachineMode[nChIdx+1].ProgramName := 'c:\TwinCAT\Cnc\Stadion.nc';
	END_IF
END_IF

IF pHmiChannel^.SetModeManual = TRUE THEN
	PlcMachineMode[nChIdx+1].Manual := pHmiChannel^.SetModeManual;
	pHmiChannel^.SetModeManual := FALSE;
END_IF

IF pHmiChannel^.SetModeMDI = TRUE THEN
	PlcMachineMode[nChIdx+1].MDI := pHmiChannel^.SetModeMDI;
	pHmiChannel^.SetModeMDI := FALSE;
END_IF

(* Channel start, stop, reset *)
IF pHmiChannel^.SetStart = TRUE THEN
	PlcMachineMode[1].Start := pHmiChannel^.SetStart;
	pHmiChannel^.SetStart := FALSE;
END_IF

IF pHmiChannel^.SetStop = TRUE THEN
	PlcMachineMode[nChIdx+1].Stop := pHmiChannel^.SetStop;
	pHmiChannel^.SetStop := FALSE;
END_IF

IF pHmiChannel^.SetReset = TRUE THEN
	PlcMachineMode[nChIdx+1].Reset := pHmiChannel^.SetReset;
	pHmiChannel^.SetReset := FALSE;
END_IF


(* Channel Error *) 
fbFlash();

IF HLI_ChannelGetState(nChan := nChIdx+1) = 6 THEN
	pHmiChannel^.Error := TRUE;
	
	IF fbFlash.bFlash = TRUE THEN
		pHmiChannel^.ErrorVis := 'Visible';
	ELSE
		pHmiChannel^.ErrorVis := 'Hidden';
	END_IF
ELSE
	pHmiChannel^.Error := FALSE;
	pHmiChannel^.ErrorVis := 'Hidden';
END_IF


(* axis data *)
FOR nAxIdx := 0 TO 10 DO
	IF	pChannel^.bahn_state.coord_r[nAxIdx].log_achs_nr_r = 0 THEN
		CONTINUE;
	END_IF

	pHmiChannel^.AxisMax := nAxIdx + 1;
	pHmiChannel^.Axis[nAxIdx].Name := pChannel^.bahn_state.coord_r[naxIdx].axis_name_r.zeichen;
	
	pAx := gpAx[naxIdx];
	pHmiChannel^.Axis[nAxIdx].actCmdPosition := pAx^.ipo_state.s_act/10000.0;		(* mm *)
	pHmiChannel^.Axis[nAxIdx].actVelo := pAx^.ipo_state.v_act/1000.0*60.0;			(* mm/min *) 
	pHmiChannel^.Axis[nAxIdx].actAcc := pAx^.ipo_state.a_act/1000.0;					(*  *)
	
	pHmiChannel^.Axis[nAxIdx].current_position_acs := pAx^.lr_state.current_position_acs_r/10000.0;		(* mm *)
	pHmiChannel^.Axis[nAxIdx].active_position_acs := pAx^.lr_state.active_position_acs_r/10000.0;		(* mm *)
	pHmiChannel^.Axis[nAxIdx].end_position_acs := pAx^.lr_state.end_position_acs_r/10000.0;				(* mm *)
	pHmiChannel^.Axis[nAxIdx].distanceToGo := pHmiChannel^.Axis[nAxIdx].end_position_acs - pHmiChannel^.Axis[nAxIdx].active_position_acs;						(* mm *)
END_FOR

END_FUNCTION_BLOCK

// ---- POUs/HMI/FB_ReadWriteFileData.TcPOU
FUNCTION_BLOCK FB_ReadWriteFileData
VAR_INPUT
	sNetId						: T_AmsNetId;		(* TwinCAT network address of the file *)
	sPathName					: T_MaxString;		(* File path and name *)
	nSeekPos						: DINT;				(* New seek pointer position *)
	bExecute						: BOOL;
	bWrite						: BOOL;				(* TRUE => Write, FALSE => Read *)
	tTimeOut						: TIME := DEFAULT_ADS_TIMEOUT;	(* Max. ADS timeout time *)
	pBuffer						: POINTER TO BYTE;
	nBufferSize					: UDINT;
END_VAR
VAR_OUTPUT
	bBusy							: BOOL;				(* TRUE => execution in progress, FALSE => execution idle *)
	bError						: BOOL;
	nErrId						: UDINT;
END_VAR
VAR
   nStep							: DWORD;
	nModeTmp						: DWORD;
	RisingEdge					: R_TRIG;
	hFile							: UINT := 0;		(* file handle *)
	fbFileOpen					: FB_FileOpen;
	fbFileClose					: FB_FileClose;
	fbFileRead					: FB_FileRead;
	fbFileWrite					: FB_FileWrite;
	fbFileSeek					: FB_FileSeek;
	bStepReady					: BOOL;
END_VAR

IF sPathName = '' THEN
	IF bWrite = FALSE THEN
		pBuffer^ := 0;
	END_IF
	RisingEdge(CLK:=FALSE);
	bBusy := FALSE;
	bError := FALSE;
	nErrId := 0;
	RETURN;
END_IF


RisingEdge(CLK:=bExecute);

CASE nStep OF
	0:		(* idle *)
		IF RisingEdge.Q THEN
			bBusy := TRUE;
			bError := FALSE;
			nErrId := 0;
			hFile := 0;
			
			IF bWrite = FALSE THEN
				nModeTmp := FOPEN_MODEREAD OR FOPEN_MODEBINARY;
			ELSE
				nModeTmp := FOPEN_MODEWRITE OR FOPEN_MODEBINARY;
			END_IF

			(*--- open file ---*)
			fbFileOpen(bExecute:=FALSE);
			fbFileOpen(sNetId:=sNetId, sPathName:=sPathName,
							nMode:=nModeTmp, ePath:=PATH_GENERIC,
							tTimeout:=tTimeOut, bExecute:=TRUE);
							
			IF NOT fbFileOpen.bBusy THEN
					bError := TRUE;
				ELSE
					bError := false;
				END_IF
							
			IF nSeekPos <> 0 THEN
				nStep := 10;
			ELSE
				nStep := 11;
			END_IF
		END_IF


	10:	(*--- wait for open finished and seek ---*)
		fbFileOpen(bExecute:=FALSE);
		IF NOT fbFileOpen.bBusy THEN
			IF fbFileOpen.bError THEN
				nErrId := fbFileOpen.nErrId;
				bError := TRUE;
				nStep := 50;
			ELSE
				hFile := fbFileOpen.hFile;

				(*--- seek file pointer ---*)
				fbFileSeek(bExecute:=FALSE);
				fbFileSeek(sNetId:=sNetId, hFile:=hFile,  
								nSeekPos:=nSeekPos, eOrigin:=SEEK_SET,
								bExecute:=TRUE, tTimeout:=tTimeOut);
				nStep := 11;
			END_IF
		END_IF
		

	11:	(*--- wait for open/seek finished and read/write---*)
		bStepReady := FALSE;
		IF nSeekPos = 0 THEN
			(*--- wait for open finished ---*)
			fbFileOpen(bExecute:=FALSE);
			IF NOT fbFileOpen.bBusy THEN
				IF fbFileOpen.bError THEN
					nErrId := fbFileOpen.nErrId;
					bError := TRUE;
					nStep := 50;
				ELSE
					hFile := fbFileOpen.hFile;
					bStepReady := TRUE;
				END_IF
			END_IF
		ELSE
			(*--- wait for seek finished ---*)
			fbFileSeek(bExecute:=FALSE);
			IF NOT fbFileSeek.bBusy THEN
				IF fbFileSeek.bError THEN
					nErrId := fbFileSeek.nErrId;
					bError := TRUE;
					nStep := 50;
				ELSE
					bStepReady := TRUE;
				END_IF
			END_IF
		END_IF
		
		IF bStepReady = TRUE THEN
			IF bWrite = FALSE THEN
				(*--- read data from file ---*)
				MEMSET(pBuffer, 0, nBufferSize);
				fbFileRead(bExecute:=FALSE);
				fbFileRead(sNetId:=sNetId, hFile:=hFile,
								pReadBuff:=pBuffer, cbReadLen:=nBufferSize,
								bExecute:=TRUE, tTimeout:=tTimeOut);
				nStep := 20;
			ELSE
				(*--- write data to file ---*)
				fbFileWrite(bExecute:=FALSE);
				fbFileWrite(sNetId:=sNetId, hFile:=hFile,
								pWriteBuff:=pBuffer, cbWriteLen:=nBufferSize,
								bExecute:=TRUE, tTimeout:=tTimeOut);
				nStep := 21;
			END_IF
		END_IF


	20:	(*--- wait for read finished and close---*)
		fbFileRead(bExecute := FALSE);
		IF NOT fbFileRead.bBusy THEN
			IF fbFileRead.bError THEN
				nErrId := fbFileRead.nErrId;
				bError := TRUE;
				nStep := 50;
			ELSE
				(*--- close the file ---*)
				fbFileClose(bExecute:=FALSE);
				fbFileClose(sNetId:=sNetId, hFile:=hFile, bExecute:=TRUE, tTimeout:=tTimeOut);
				nStep := 30;
			END_IF
		END_IF


	21:	(*--- wait for write finished and close ---*)
		fbFileWrite(bExecute:=FALSE);
		IF NOT fbFileWrite.bBusy THEN
			IF fbFileWrite.bError THEN
				nErrId := fbFileWrite.nErrId;
				bError := TRUE;
				nStep := 50;
			ELSE
				(*--- close the file ---*)
				fbFileClose(bExecute:=FALSE);
				fbFileClose(sNetId:=sNetId, hFile:=hFile, bExecute:=TRUE, tTimeout:=tTimeOut);
				nStep := 30;
			END_IF
		END_IF


	30:	(*--- wait for close finished ---*)
		fbFileClose(bExecute:=FALSE);
		IF NOT fbFileClose.bBusy THEN
			IF fbFileClose.bError THEN
				nErrId := fbFileClose.nErrId;
				bError := TRUE;
				nStep := 50;
			ELSE
				hFile := 0;
				nStep := 0;			(* ready *)
				bBusy := FALSE;
			END_IF
		END_IF

	50:	(*--- Error ---*)
		IF (hFile <> 0) THEN
			(*--- try close the file ---*)
			fbFileClose(bExecute:=FALSE);
			fbFileClose(sNetId:=sNetId, hFile:=hFile, bExecute:=TRUE, tTimeout:=tTimeOut);
			nStep := 30;		(* wait for close *)
		ELSE
			nStep := 0;			(* ready *)
			bBusy := FALSE;
		END_IF

END_CASE

END_FUNCTION_BLOCK

// ---- POUs/HMI/FB_ReadTechnoGFunc.TcPOU
FUNCTION_BLOCK FB_ReadTechnoGFunc
VAR_INPUT
   sNetId               : T_AmsNetId;
   nPort                : T_AmsPort := 553;
   nIdxGrp              : UDINT;
   nIdxOffs             : UDINT;
	nLen						: UDINT;
   bStart               : BOOL;
	pStr						: POINTER TO STRING;
END_VAR
VAR_OUTPUT
   bBusy                : BOOL;
   bErr                 : BOOL;
END_VAR
VAR
   fbRead               : ADSREAD;
   bStarted             : BOOL;
   destArr               : ARRAY[0..40] OF INT;
	i							: INT;
	tmp						: STRING;
END_VAR

(* ========================================================= *)
(*     FB: FB_ReadTechnoGFunc                                *)
(* --------------------------------------------------------- *)
(*   Desc: Reads the technology information                  *)
(*       : from the CNC                                      *)
(* Author: MK                                                *)
(*   Date: 21.12.2011                                        *)
(*   Rev.: 1.0                                               *)
(* ========================================================= *)


IF bStart = TRUE AND bStarted = FALSE THEN
	bStarted := TRUE;
	bErr := FALSE;
	bBusy := TRUE;
END_IF

IF bStarted THEN
   fbRead(NetID:=sNetId, Port:=nPort, IdxGrp:=nIdxGrp, IdxOffs:=nIdxOffs,
         LEN:=nLen, DestAddr:=ADR(destArr), READ:=bStarted, TMOUT:=DEFAULT_ADS_TIMEOUT);
   IF NOT fbRead.Busy THEN
      IF fbRead.Err THEN
         bErr := TRUE;
		ELSE
			tmp := '';
			FOR i:=0 TO 36 DO
				IF destArr[i] <> -1 THEN
					tmp := CONCAT(tmp, 'G');
					tmp := CONCAT(tmp, INT_TO_STRING(destArr[i]));
					tmp := CONCAT(tmp, ' ');
		      END_IF
			END_FOR
			pStr^ := tmp;
      END_IF
      fbRead(READ := FALSE);
      bStarted := FALSE;
      bBusy := FALSE;
   END_IF
END_IF

END_FUNCTION_BLOCK

// ---- POUs/HMI/FB_ReadTechnoMFunc.TcPOU
FUNCTION_BLOCK FB_ReadTechnoMFunc
VAR_INPUT
   sNetId               : T_AmsNetId;
   nPort                : T_AmsPort := 553;
   nIdxGrp              : UDINT;
   nIdxOffs             : UDINT;
	nLen						: UDINT;
   bStart               : BOOL;
	pStr						: POINTER TO STRING;
END_VAR
VAR_OUTPUT
   bBusy                : BOOL;
   bErr                 : BOOL;
END_VAR
VAR
   fbRead               : ADSREAD;
   bStarted             : BOOL;
   destArr             : ARRAY[0..40] OF UDINT;
	i							: UDINT;
	nMax						: UDINT;
	tmp						: STRING;
END_VAR

(* ========================================================= *)
(*     FB: FB_ReadTechnoMFunc                                *)
(* --------------------------------------------------------- *)
(*   Desc: Reads the technology information                  *)
(*       : from the CNC                                      *)
(* Author: MK                                                *)
(*   Date: 21.12.2011                                        *)
(*   Rev.: 1.0                                               *)
(* ========================================================= *)


IF bStart = TRUE AND bStarted = FALSE THEN
	bStarted := TRUE;
	bErr := FALSE;
	bBusy := TRUE;
END_IF

IF bStarted THEN
   fbRead(NetID:=sNetId, Port:=nPort, IdxGrp:=nIdxGrp, IdxOffs:=nIdxOffs,
         LEN:=nLen, DestAddr:=ADR(destArr), READ:=bStarted, TMOUT:=DEFAULT_ADS_TIMEOUT);
   IF NOT fbRead.Busy THEN
      IF fbRead.Err THEN
         bErr := TRUE;
		ELSE
			tmp := '';
			nMax := destArr[0];
			FOR i:=1 TO nMax DO
				IF destArr[i] <> -1 THEN
					tmp := CONCAT(tmp, 'M');
					tmp := CONCAT(tmp, UDINT_TO_STRING(destArr[i]));
					tmp := CONCAT(tmp, ' ');
		      END_IF
			END_FOR
			pStr^ := tmp;
      END_IF
      fbRead(READ := FALSE);
      bStarted := FALSE;
      bBusy := FALSE;
   END_IF
END_IF

END_FUNCTION_BLOCK

// ---- POUs/HMI/FB_ReadTechnoTFunc.TcPOU
FUNCTION_BLOCK FB_ReadTechnoTFunc
VAR_INPUT
   sNetId               : T_AmsNetId;
   nPort                : T_AmsPort := 553;
   nIdxGrp              : UDINT;
   nIdxOffs             : UDINT;
	nLen						: UDINT;
   bStart               : BOOL;
	pStr						: POINTER TO STRING;
END_VAR
VAR_OUTPUT
   bBusy                : BOOL;
   bErr                 : BOOL;
END_VAR
VAR
   fbRead               : ADSREAD;
   bStarted             : BOOL;
   dest                 : UDINT;
	i							: INT;
	tmp						: STRING;
END_VAR

(* ========================================================= *)
(*     FB: FB_ReadTechnoTFunc                                *)
(* --------------------------------------------------------- *)
(*   Desc: Reads the technology information                  *)
(*       : from the CNC                                      *)
(* Author: MK                                                *)
(*   Date: 21.12.2011                                        *)
(*   Rev.: 1.0                                               *)
(* ========================================================= *)


IF bStart = TRUE AND bStarted = FALSE THEN
	bStarted := TRUE;
	bErr := FALSE;
	bBusy := TRUE;
END_IF

IF bStarted THEN
   fbRead(NetID:=sNetId, Port:=nPort, IdxGrp:=nIdxGrp, IdxOffs:=nIdxOffs,
         LEN:=nLen, DestAddr:=ADR(dest), READ:=bStarted, TMOUT:=DEFAULT_ADS_TIMEOUT);
   IF NOT fbRead.Busy THEN
      IF fbRead.Err THEN
         bErr := TRUE;
		ELSE
			tmp := 'T';
			tmp := CONCAT(tmp, UDINT_TO_STRING(dest));
			pStr^ := tmp;
      END_IF
      fbRead(READ := FALSE);
      bStarted := FALSE;
      bBusy := FALSE;
   END_IF
END_IF

END_FUNCTION_BLOCK

// ---- POUs/General/FB_Flash.TcPOU
FUNCTION_BLOCK FB_Flash
VAR_INPUT
	tiTime_On							: TIME := T#0.5S;		(* Zeitwert für Blinkbit ein *)
	tiTime_Off							: TIME := T#0.5s;		(* Zeitwert für Blinkbit aus *)
END_VAR
VAR_OUTPUT
	bFlash								: BOOL;					(* Blinkbit *)
END_VAR
VAR
	tnTimer_ON							: TON;
	tnTimer_OFF							: TON;
END_VAR

tnTimer_OFF(IN:=tnTimer_ON.Q, PT:=tiTime_On);
tnTimer_ON(IN:=NOT tnTimer_OFF.Q, PT:=tiTime_Off);
bFlash := tnTimer_ON.Q;

END_FUNCTION_BLOCK

// ---- POUs/CNC/F3_Control/HLI_ChannelGetState.TcPOU
FUNCTION HLI_ChannelGetState : DWORD
VAR_INPUT
	nChan					: UDINT;			(* Number of channel *)
END_VAR
VAR
	nHliChIdx			: UDINT;
END_VAR

(* ========================================================= *)
(*    FUN: HLI_ChannelGetState                               *)
(* --------------------------------------------------------- *)
(*   Desc:                                                   *)
(* Author: MK                                                *)
(*   Date: 21.12.2011                                        *)
(*   Rev.: 1.0                                               *)
(* ========================================================= *)


nHliChIdx := nChan - 1;

IF nChan <= 0 OR gNrCh < nChan OR			(* check for channel no *)
	gpCh[nHliChIdx] = 0 THEN					(* check for zero pointer *)
	HLI_ChannelGetState := 0;
	RETURN; (* e x i t *)
END_IF

(* if the stop button from the HMI is selected the request is set *)
HLI_ChannelGetState := gpCh[nHliChIdx]^.channel_mc_control.mode_and_state.state_r.state;

END_FUNCTION

// ---- POUs/General/WritePersistentData.TcPOU
PROGRAM WritePersistentData
VAR
	bWriteData							: BOOL;
	fbWritePersistentData			: FB_WritePersistentData;
	rtWriteData							: R_TRIG;
	bIsActive							: BOOL;

	Busy									: BOOL;
	ERR									: BOOL;
	ERRID									: UDINT;
	fbFlash1								: FB_Flash;
	bGo									: BOOL := false;
END_VAR


fbFlash1(tiTime_On := T#10MS, tiTime_Off := T#10MS);
bWriteData := fbFlash1.bFlash and bGo;

rtWriteData(CLK:=bWriteData);
IF rtWriteData.Q THEN
	bIsActive := TRUE;
END_IF


IF bIsActive THEN
	fbWritePersistentData(NETID:='', PORT:=851, START:=bIsActive, TMOUT:=T#1s, MODE := SPDM_2PASS);
	IF fbWritePersistentData.BUSY = FALSE THEN
		fbWritePersistentData(START:=FALSE);
		bIsActive := FALSE;
	END_IF
END_IF

Busy := fbWritePersistentData.BUSY;
ERR := fbWritePersistentData.ERR;
ERRID := fbWritePersistentData.ERRID;

END_PROGRAM

// ---- POUs/Messages/ShowMessages.TcPOU
PROGRAM ShowMessages
VAR
	SimpleEventLog1		: FB_SimpleEventLog;
	SimpleEventLog2		: FB_SimpleEventLog;
	SimpleEventLog3		: FB_SimpleEventLog;
	SimpleEventLog4		: FB_SimpleEventLog;

	bStart					: BOOL;

	bClear					: BOOL := TRUE;
	ClearEvents				: ADSCLEAREVENTS;

	bSetMsg1					: BOOL;
	bSetMsg2					: BOOL;
END_VAR

(* ----------------------------------------------------------
	Clears all active and logged events at startup.
	Should only be used at the startup sequence!
	During PLC runtime cycle each event has to be handled with
	set event, acknowledge event and or quit event!
	Don't use ClearEvents in any other case!!!
   ---------------------------------------------------------- *)
IF bClear THEN
  ClearEvents(NetID:='', bClear:=TRUE, iMode:=TCEVENTLOGIOFFS_CLEARALL, tTimeout:= t#1s);
  bClear := FALSE;
ELSE
  ClearEvents(bClear:=FALSE);
END_IF;


(* ----------------------------------------------------------
	Shows how to display messages.
	At startup the different message lists are set up.
	If new message lists are added, don't forget to restart again!

	The different message classes are listed below.

	TCEVENTCLASS_NONE				:=0,	 No class
	TCEVENTCLASS_MAINTENANCE	:=1,	 Maintenance hint
	TCEVENTCLASS_MESSAGE			:=2,	 Message
	TCEVENTCLASS_HINT				:=3,	 Hint
	TCEVENTCLASS_STATEINFO		:=4,	 State information
	TCEVENTCLASS_INSTRUCTION	:=5,	 Instruction
	TCEVENTCLASS_WARNING			:=6,	 Warning
	TCEVENTCLASS_ALARM			:=7,	 Alarm
	TCEVENTCLASS_PARAMERROR		:=8	 Parameter error
   ---------------------------------------------------------- *)

IF NOT bStart THEN
	bStart := TRUE;
	SimpleEventLog1(Init				:= TRUE,
						SourceId			:= 50,
						Class				:= TCEVENTCLASS_WARNING,
						QuitRequired	:= FALSE,
						adrAlarmArray	:= ADR(MSGList1),
						adrQuitArray	:= ADR(MSGListQuit1));

	SimpleEventLog2(Init				:= TRUE,
						SourceId			:= 51,
						Class				:= TCEVENTCLASS_ALARM,
						QuitRequired	:= FALSE,
						adrAlarmArray	:= ADR(MSGList2),
						adrQuitArray	:= ADR(MSGListQuit2));

	SimpleEventLog3(Init				:= TRUE,
						SourceId			:= 52,
						Class				:= TCEVENTCLASS_INSTRUCTION,
						QuitRequired	:= FALSE,
						adrAlarmArray	:= ADR(MSGList3),
						adrQuitArray	:= ADR(MSGListQuit3));

	SimpleEventLog4(Init				:= TRUE,
						SourceId			:= 1000,
						Class				:= TCEVENTCLASS_ALARM,
						QuitRequired	:= FALSE,
						adrAlarmArray	:= ADR(MSGList4),
						adrQuitArray	:= ADR(MSGListQuit4));
ELSE
	SimpleEventLog1(Init:=FALSE);
	SimpleEventLog2(Init:=FALSE);
	SimpleEventLog3(Init:=FALSE);
	SimpleEventLog4(Init:=FALSE);
END_IF

END_PROGRAM

// ---- POUs/Messages/FB_SimpleEventLog.TcPOU
(*****************************************************************************************
Name:				FB_SimpleEventLog
Date:				13.10.2004
Author:			Dirk Nordberg (BECKHOFF INDUSTRIE ELEKTRONIK)

Description: Function block to control the EventLogger
	Messages can be activated or deactivated through an array of bool.
	The subscription of the array is equivalent to EventID from EventLogger.
	Funtion block will be initialized with Init flag, then the busy flag is set true. 

	Revision:	1.3
	History:		13.10.2004	Ng	start coding
					17.04.2005	MK	runtime optimized
					07.07.2005	MK	short puls BF
*****************************************************************************************)
FUNCTION_BLOCK FB_SimpleEventLog
VAR_INPUT
	Init				: BOOL;				(* Rising flag starts the initialization *)
	SourceId			: UINT;				(* Number of the source Id *)
	Class				: UINT;				(* Alarm error class *)
	QuitRequired	: BOOL;				(* Activate or deaktivate confirmation *)
	adrAlarmArray	: POINTER TO BOOL;(* Adress of the array for the messages *)
												(* ...with constant boundaries ARRAY_LBOUND to ARRAY_UBOUND for array size *)
	adrQuitArray	: POINTER TO BOOL;(* Adress of the array for the confirmations	*)
												(* ...with constant boundaries ARRAY_LBOUND to ARRAY_UBOUND for array size *)
END_VAR
VAR_OUTPUT
	Busy				: BOOL;
	Err 				: BOOL;
	ErrId			 	: UDINT;
END_VAR
VAR CONSTANT
	ARRAY_LBOUND				: INT := FIRST_MESSAGE;
	ARRAY_UBOUND				: INT := LAST_MESSAGE;
	TCEVENTDATAFORMATSTRING	: STRING := ' ';
	STATE_INIT					: INT := 0;
	STATE_IDLE					: INT := 1;
	STATE_RESET_EVENT			: INT := 2;
	STATE_QUIT_EVENT			: INT := 3;
	STATE_RESET_END			: INT := 4;
	STATE_WAIT					: INT := 5;
END_VAR
VAR
	state					: INT;
(*{flag nowatch on }*)
	bReady				: BOOL := TRUE;
	nMsgHasChanged		: DINT;
	bEvtState			: ARRAY [ARRAY_LBOUND..ARRAY_UBOUND] OF BOOL;
	event					: ARRAY [ARRAY_LBOUND..ARRAY_UBOUND] OF ADSLOGEVENT;
	idx					: INT;
	CfgEvent				: TcEvent;
	bWait					: BOOL;
	ptAlarm				: POINTER TO BOOL;
	ptQuit				: POINTER TO BOOL;
	RT_Init				: R_TRIG;
(*{flag off}*)
END_VAR


nMsgHasChanged := MEMCMP(ADR(bEvtState), adrAlarmArray, SIZEOF(bEvtState));
RT_Init(CLK:=Init);

CASE State OF
	STATE_INIT:		(* Set the parameter for TcEvent *)
		Err := FALSE;
		ErrId :=0;
		Busy := FALSE;
		CfgEvent.Prio := 0;
		CfgEvent.DataFormatStrAddress := ADR(TCEVENTDATAFORMATSTRING);
		CfgEvent.Flags := TCEVENTFLAG_LOG OR TCEVENTFLAG_SRCID;
		CfgEvent.StreamType := TCEVENTSTREAM_SIMPLE;
		CfgEvent.ProgId := 'TcEventFormatter.TcXmlFormatter';
		CfgEvent.Prio := 1;
		CfgEvent.SourceId := SourceId;
		CfgEvent.Class := Class ;
		CfgEvent.bQuitRequired := QuitRequired;
		FOR idx := ARRAY_LBOUND TO ARRAY_UBOUND BY 1 DO
			CfgEvent.Id := idx;
			event[idx](NETID:='', PORT:=110, Event:=FALSE , EventQuit:=FALSE,
				 EventConfigData:=CfgEvent, FbCleanup:=FALSE, TMOUT:=t#1s);
		END_FOR;
		State := STATE_IDLE;

	STATE_IDLE:
		(* nothing to do *)
		IF nMsgHasChanged = 0
			AND bReady = TRUE
			AND NOT RT_Init.Q THEN
			RETURN;
		END_IF

		IF adrAlarmArray <> 0 THEN
			ptAlarm := adrAlarmArray;
			IF CfgEvent.bQuitRequired AND adrQuitArray <> 0 THEN
				ptQuit := adrQuitArray;
				FOR idx := ARRAY_LBOUND TO ARRAY_UBOUND BY 1 DO
					event[idx](Event:=ptAlarm^, EventQuit:=ptQuit^);
					ptAlarm := ptAlarm + 1;
					ptQuit := ptQuit + 1;
				END_FOR;
			ELSE
				bReady := TRUE;
				FOR idx := ARRAY_LBOUND TO ARRAY_UBOUND BY 1 DO
					event[idx](Event:=ptAlarm^);
					IF (NOT(ptAlarm^ = TRUE
							AND event[idx].Event = TRUE		(* event is set/on *)
							AND event[idx].Quit = FALSE
							AND event[idx].EventState = TCEVENTSTATE_SIGNALED)
						AND NOT (ptAlarm^ = FALSE
							AND event[idx].Event = FALSE		(* event is reset/off *)
							AND event[idx].Quit = TRUE
							AND event[idx].EventState = TCEVENTSTATE_INVALID)) THEN
						bReady := FALSE;
					END_IF
					ptAlarm := ptAlarm + 1;
				END_FOR;

				(* copy the status *)
				IF bReady THEN
					MEMCPY(ADR(bEvtState), adrAlarmArray, SIZEOF(bEvtState));
				END_IF

			END_IF
		END_IF

		IF RT_Init.Q THEN
			Busy := TRUE;
			State := STATE_RESET_EVENT;
		END_IF

	STATE_RESET_EVENT:(*---------------------------------- clear messages ----------------------------------------*)
		FOR idx := ARRAY_LBOUND TO ARRAY_UBOUND BY 1 DO
			IF event[idx].EventState = TCEVENTSTATE_SIGNALED THEN
				event[idx](Event:=FALSE, EventQuit:= FALSE, FbCleanup:= FALSE, TMOUT:= t#1s);
				IF event[idx].Err THEN
					Err := TRUE;
					ErrId := event[idx].ErrId;
					IF event[idx].ErrId = 1282 THEN	(* Message Router: mailbox full *)
						event[idx](Event:=FALSE, EventQuit:= FALSE, FbCleanup:= FALSE);
						RETURN;
					END_IF
				END_IF
			END_IF;
		END_FOR;
		State := STATE_QUIT_EVENT;

	STATE_QUIT_EVENT:(*---------------------------------- quit messages ----------------------------------------*)
		FOR idx := ARRAY_LBOUND TO ARRAY_UBOUND BY 1 DO
			IF event[idx].EventState = TCEVENTSTATE_SIGNALED THEN
				event[idx](Event:=FALSE, EventQuit:= TRUE, FbCleanup:= FALSE, TMOUT:= t#1s);
				IF event[idx].Err THEN
					Err := TRUE;
					ErrId := event[idx].ErrId;
					IF event[idx].ErrId = 1282 THEN	(* Message Router: mailbox full *)
						event[idx](Event:=FALSE, EventQuit:= FALSE, FbCleanup:= FALSE);
						RETURN;
					END_IF
				END_IF
			END_IF;
		END_FOR;
		State := STATE_RESET_END;

	STATE_RESET_END:
		bWait := FALSE;
		FOR idx := ARRAY_LBOUND TO ARRAY_UBOUND BY 1 DO
			event[idx](Event:=FALSE, EventQuit:= FALSE, FbCleanup:= FALSE);
			IF event[idx].EventState = TCEVENTSTATE_SIGNALED THEN
				bWait := TRUE;
			END_IF
		END_FOR;
		IF NOT bWait THEN
			State := STATE_INIT;
		END_IF

END_CASE

END_FUNCTION_BLOCK

// ---- POUs/CNC/F9_Misc/MySystemTime.TcPOU
PROGRAM MySystemTime
VAR
	nState								: INT;
	fbGetTime							: NT_GetTime;
	tonGetTime							: TON;
	bSystemTimeValid					: BOOL := FALSE;
	bFirstCycle							: BOOL;

	ptBaseTime							: TIME := t#1000ms;
	ptTime								: TIME := t#1000ms;
	dtSystemTime						: DT;
	stSystemTime						: TIMESTRUCT;
	sTime 								: STRING;		(*long date, time string*)
	sShortTime 							: STRING;		(*short time string*)
	sShortDate 							: STRING;		(*short date string*)
	nDayShortDate						: WORD;

	(* time zone information *)
	wHour									: WORD := 99;
	tzID									: E_TimeZoneID := eTimeZoneID_Invalid;
																(*	eTimeZoneID_Invalid := -1,
																	eTimeZoneID_Unknown := 0,
																	eTimeZoneID_Standard := 1,
																	eTimeZoneID_Daylight := 2 *)
	fbGetTimeZoneInformation		: FB_GetTimeZoneInformation;
END_VAR

(* Read the time *)

IF bFirstCycle = FALSE THEN
	bFirstCycle := TRUE;
	(* 970 = 1000 - 30 bei 10ms, 930 = 1000 - 60 bei 20ms ??? 921-940 *)
	ptBaseTime := T#1000MS - UDINT_TO_TIME(3 * TwinCAT_SystemInfoVarList._TaskInfo[1].CycleTime/10000);
	ptTime := ptBaseTime;
END_IF


CASE nState OF
	0:
		tonGetTime(IN := TRUE, PT := ptTime);
		IF tonGetTime.Q THEN
			tonGetTime(IN := FALSE);
			nState := 10;
		END_IF

	10:
		fbGetTime(START := TRUE);
		IF fbGetTime.BUSY = FALSE THEN
			stSystemTime := fbGetTime.TIMESTR;
			dtSystemTime := SYSTEMTIME_TO_DT(fbGetTime.TIMESTR);
			fbGetTime(START := FALSE);
			sTime := SYSTEMTIME_TO_STRING(stSystemTime);
			sShortTime := MID(STR:=sTime, LEN:=8, POS:=12);

			(* build short date string *)
			IF nDayShortDate <> MySystemTime.stSystemTime.wDay THEN
				nDayShortDate := MySystemTime.stSystemTime.wDay;
				(* day *)
				IF MySystemTime.stSystemTime.wDay < 10 THEN
					sShortDate := CONCAT(STR1:='0', STR2:=DWORD_TO_STRING(MySystemTime.stSystemTime.wDay));
				ELSE
					sShortDate := DWORD_TO_STRING(MySystemTime.stSystemTime.wDay);
				END_IF
				sShortDate := CONCAT(STR1:=sShortDate, STR2:='.');
				(* month *)
				IF MySystemTime.stSystemTime.wMonth < 10 THEN
					sShortDate := CONCAT(STR1:=sShortDate, STR2:='0');
					sShortDate := CONCAT(STR1:=sShortDate, STR2:=DWORD_TO_STRING(MySystemTime.stSystemTime.wMonth));
				ELSE
					sShortDate := CONCAT(STR1:=sShortDate, STR2:=DWORD_TO_STRING(MySystemTime.stSystemTime.wMonth));
				END_IF
				(* year *)
				sShortDate := CONCAT(STR1:=sShortDate, STR2:='.');
				sShortDate := CONCAT(STR1:=sShortDate, STR2:=DWORD_TO_STRING(MySystemTime.stSystemTime.wYear));
			END_IF

			bSystemTimeValid := TRUE;
			nState := 0;

			IF stSystemTime.wMilliseconds > 30 THEN
				ptTime := ptBaseTime - t#20ms;
			ELSIF stSystemTime.wMilliseconds < 7 THEN
				ptTime := ptBaseTime + T#20MS;
			ELSE
				ptTime := ptBaseTime;
			END_IF
		END_IF

END_CASE


(* get time zone information, summer/winter, only once a day *)
IF MySystemTime.stSystemTime.wHour <> wHour THEN
	IF MySystemTime.stSystemTime.wHour = 4 OR wHour = 99 THEN

		fbGetTimeZoneInformation(bExecute := TRUE);
		IF fbGetTimeZoneInformation.bBusy = FALSE THEN
			fbGetTimeZoneInformation(bExecute := FALSE);
			tzID := fbGetTimeZoneInformation.tzID;
			wHour := MySystemTime.stSystemTime.wHour;
		END_IF

	ELSE
		wHour := MySystemTime.stSystemTime.wHour;
	END_IF
END_IF

END_PROGRAM

// ---- POUs/CNC/F1_Init/HLI_Init.TcPOU
PROGRAM HLI_Init
VAR
	HliInterface		: MCV_HliInterface;
	tool					: CncToolControl;
	MessageOutput		: R_TRIG;
	
	bFirstCycle			: BOOL := TRUE;
	bInitHLI				: BOOL;
END_VAR

(* ========================================================= *)
(*    PRG: HLI_Init                                          *)
(* --------------------------------------------------------- *)
(*   Desc:                                                   *)
(* Author: MK                                                *)
(*   Date: 21.12.2011                                        *)
(*   Rev.: 1.0                                               *)
(* ========================================================= *)


(* Init Tool Configuration structures *)
tool.HandleExternalToolData();
tool.SetToolData();


IF NOT bInitHLI THEN
	HliInterface();
	IF HliInterface.Initialized = TRUE THEN
		bInitHLI := TRUE;
	END_IF
END_IF

IF HliInterface.Initialized = TRUE AND HliInterface.Error = FALSE THEN
	(* User initialization, used during start of PLC once *)
	IF CncSystem.bUserInitDone = FALSE THEN
		(* Initialisierungen auf dem HLI-Interface *)
		CncSystem.bUserInitDone := HLI_UserInitialisation();

		ADSLOG(strMsg:='High Level Interfaces initialized: %s', nDINT:=0, strArg:='');
	END_IF

	(* initialization finished *)
	CNCSystem.bHLIInit := TRUE;
ELSE
	MessageOutput(CLK:=HliInterface.Error);
	IF HliInterface.Error = TRUE	THEN
		(* Fehler beim Initialisieren des HLI *)
		IF MessageOutput.Q THEN
			ADSLOGDINT(	msgCtrlMask := ADSLOG_MSGTYPE_ERROR OR
												ADSLOG_MSGTYPE_MSGBOX OR
												ADSLOG_MSGTYPE_LOG,
							msgFmtStr := 'Fehler beim Initialisieren des HLI-Interfaces Fehlercode: %d',
							dintArg := HliInterface.ErrorID);
		END_IF
		CNCSystem.nInitErrorId := HliInterface.ErrorID;
		CNCSystem.bInitError := TRUE;
	END_IF;
END_IF

END_PROGRAM

// ---- POUs/CNC/F1_Init/CncToolControl.TcPOU
FUNCTION_BLOCK CncToolControl
VAR_INPUT
END_VAR
VAR_OUTPUT
	bInitialized			: BOOL;
END_VAR
VAR
END_VAR

METHOD PUBLIC SetToolData
VAR_INPUT
END_VAR
VAR
	i						: UINT;
	pToolData			: POINTER TO ST_ToolData;
END_VAR
(* ========================================================= *)
(*    PRG: HLI_SetToolData                                   *)
(* --------------------------------------------------------- *)
(*   Desc:                                                   *)
(* Author: MK                                                *)
(*   Date: 11.03.2015                                        *)
(*   Rev.: 1.2                                               *)
(* ========================================================= *)


(* init basic tool structure *)
IF TwinCAT_SystemInfoVarList._TaskInfo[1].FirstCycle OR PlcToolManagement.ToolDataActive = TRUE THEN
	(* last tool indicates system tool change *)
	PlcToolManagement.ToolDataActive := FALSE;

	(* adapt tool parameter settings here *)
	FOR i := 1 TO MAX_TOOLS DO
		(*CncSystem.Tool[i].tool_life.dist_used := 0.0;
		CncSystem.Tool[i].tool_life.time_used := 0.0; *)

		pToolData := ADR(PlcToolManagement.ToolData[i]);
		CncSystem.Tool[i].tool_desc.tool_id.basic	:= i;
		CNCSystem.Tool[i].tool_desc.valid := (pToolData^.ToolLocked = 0);
		CncSystem.Tool[i].tool_desc.tool_id.sister := pToolData^.SisterTool;
		(*CncSystem.Tool[i].tool_desc.tool_id.sister_valid := TRUE;*)
		CNCSystem.Tool[i].tool_desc.radius := LREAL_TO_DINT((pToolData^.Radius + pToolData^.DeltaRadius) * 10000.0);
		CNCSystem.Tool[i].tool_desc.laenge := LREAL_TO_DINT((pToolData^.Length + pToolData^.DeltaLength) * 10000.0);
		CNCSystem.Tool[i].tool_desc.ax_versatz[0] := LREAL_TO_DINT(pToolData^.Param1 * 10000.0);
		CNCSystem.Tool[i].tool_desc.ax_versatz[1] := LREAL_TO_DINT(pToolData^.Param2 * 10000.0);
		CNCSystem.Tool[i].tool_desc.ax_versatz[2] := LREAL_TO_DINT(pToolData^.Param3 * 10000.0);
		CncSystem.Tool[i].tool_desc.param[0] := pToolData^.Param4 * 10000.0;
		CncSystem.Tool[i].tool_desc.param[1] := pToolData^.Param5 * 10000.0;
		CncSystem.Tool[i].tool_desc.param[2] := pToolData^.Param6 * 10000.0;
		CncSystem.Tool[i].tool_desc.param[3] := pToolData^.Param7 * 10000.0;
	END_FOR
	
	bInitialized := TRUE;
END_IF
END_METHOD

METHOD PUBLIC HandleExternalToolData
VAR
	BasicToolId			: DINT;
	(*ToolId				: CNC_TOOL_ID;*)

	pToolId				: POINTER TO CNC_TOOL_ID;
	pToolReq				: POINTER TO CNC_TOOL_REQUEST_IN;
	pToolLife			: POINTER TO CNC_TOOL_DATA_IN;

	RInd					: ADSRDWRTIND;
	RRes					: ADSRDWRTRES;
	bRes					: BOOL;
	i						: INT;
END_VAR
(* ---------------------*----------------------------------|------------------------------------------------------- *)
(* PURPOSE: HandleExternalToolData                                                                                  *)
(*          used for tool change and tool live between CNC and PLC                                                  *)
(*                                                                                                                  *)
(* SCOPE:                                                                                                           *)
(*                                                                                                                  *)
(*                                                                                                                  *)
(* REMARKS:                                                                                                         *)
(*                                                                                                                  *)
(*                                                                                                                  *)
(* AUTHOR:              VERSION     DATE                   CHECKED FROM      DATE     STATUS                        *)
(*    MK                1.0         21.12.2011                                                                      *)
(*                                                                                                                  *)
(* ---------------------*----------------------------------|------------------------------------------------------- *)

(*
 ATTENTION: These Indications are only sent by the CNC if the CNC channel is configured accordingly:
In the SDA-MDS parammeter list the following parameters must be set:
- ext_wzv_vorhanden    1   -> (external tool managment present) Tool requests D<i> are sent TO external tool data manager
- einrechnen_mit_t     0/1 -> programming T<i> implies a programmed D<i>
- tool_life_to_wzv     1   -> send tool data life parameters TO external tool data manager IF tool is changed.
- t_info_to_wzv        1   -> send tool to external tool data manager IF tool is programmed.

CNC_TOOL_ID :
	basic					: DINT;
	sister				: DINT;
	variant				: DINT;
	sister_valid		: BOOL;
	variant_valid		: BOOL;
	res1					: BYTE;
	res2					: BYTE;
CNC_TOOL_REQUEST_IN :
	id						: CNC_TOOL_ID; 		(* tool id of requested tool *)
	act_t_nr				: DINT;					(* actual t number in nc kernel *)
	act_d_nr				: CNC_TOOL_ID; 		(* actual tool id (d-number) in the nc kernel *)
	param					: ARRAY [1..60] OF LREAL;
CNC_TOOL_DESC :
	tool_id				: CNC_TOOL_ID;
	laenge				: DINT;
	radius				: DINT;
	ax_versatz			: ARRAY [1..32] OF DINT;
	kopf_versatz		: ARRAY [1..28] OF DINT;
	mass_einheit		: UINT;
	typ					: UINT;
	srk_lage				: UINT;
	kin_id				: UINT;
	log_ax_nr_spdl		: UINT;
	tool_fixed			: BOOL;
	valid					: BOOL;
	res					: ARRAY [1..4] OF BYTE;
	param					: ARRAY [1..60] OF LREAL;
	vb_min				: LREAL;
	vb_max				: LREAL;
	a_max					: LREAL;
*)


(* Init Tool Configuration *)
bRes := FALSE;
Rind();

IF RInd.VALID THEN
	(* initialize response *)
	RRes.NETID		:= '';
	RRes.PORT		:= RInd.PORT;
	RRes.INVOKEID	:= RInd.INVOKEID;
	bRes := TRUE;

	(* Since there is only one ADSRDWRTIND possible per PLC task *)
	(* all indications have to be handled in one place *)
	(* To distinguish between several possible request types *)
	(* the indexgroup of the ADSRDWRTIND is used *)

	(* CNC tool data request with T<i>, during NC program decoding *)
	IF RInd.IDXGRP = ADS_IGRP_TOOL_INFO_WRITE THEN (* 16#80040000 *)

		(* Tool data request from CNC *)
		pToolId		:= RInd.DATAADDR;
		BasicToolId	:= pToolId^.basic;

		IF BasicToolId <= MAX_TOOLS THEN
			(* Tool id in valid range *)
			RRes.LEN			:= SIZEOF(pToolId^);
			RRes.DATAADDR	:= pToolId;
			RRes.RESULT		:= ADS_RDWRT_IND_NO_ERROR;

			(*
			RRes.RESULT		:= 0;
			RRes.LEN			:= SIZEOF(CncSystem.Tool[1]);
			RRes.DATAADDR	:= ADR(CncSystem.Tool[ToolId.basic]); *)
		ELSE
			RRes.RESULT		:= WZV_TOOL_ID_BASIC_INVALID;
		END_IF

	(* CNC tool data request with D<i> *)
	ELSIF RInd.IDXGRP = ADS_IGRP_TOOL_DESC_READ THEN

		(* Tool data request from CNC *)
		pToolReq		:= RInd.DATAADDR;
		BasicToolId	:= pToolReq^.id.basic;

		IF BasicToolId <= MAX_TOOLS THEN
			(* transmit tool data in the response *)
			RRes.LEN			:= SIZEOF(CncSystem.Tool[1].tool_desc);
			RRes.DATAADDR	:= ADR(CncSystem.Tool[BasicToolId].tool_desc);
			RRes.RESULT		:= ADS_RDWRT_IND_NO_ERROR;
		ELSE
			(* Tool not present *)
			RRes.LEN			:= 0;
			RRes.DATAADDR	:= 0;
			RRes.RESULT		:= WZV_TOOL_ID_BASIC_INVALID;
		END_IF

	(*----- CNC tool life -----*)
	(* CNC actualize tool life data after tool change T<i> *)
	ELSIF RInd.IDXGRP = ADS_IGRP_TOOL_LIFE_DATA_WRITE THEN

		(* CNC writes tool life data *)
		pToolLife	:= RInd.DATAADDR;
		BasicToolId	:= pToolLife^.tool_id.basic;

		(* no data transmitted in the response *)
		RRes.LEN			:= 0;
		RRes.DATAADDR	:= 0;

		IF BasicToolId <= MAX_TOOLS THEN
			(* actualize tool life data *)
			CncSystem.Tool[BasicToolId].tool_life.dist_used := CncSystem.Tool[BasicToolId].tool_life.dist_used
													+ pToolLife^.dist_used;
			CncSystem.Tool[BasicToolId].tool_life.time_used := CncSystem.Tool[BasicToolId].tool_life.time_used
													+ pToolLife^.time_used;

			(* tool life data to tool management *)
			PlcToolManagement.ToolLife.tool_id := BasicToolId;
			PlcToolManagement.ToolLife.dist_used := pToolLife^.dist_used;
			PlcToolManagement.ToolLife.time_used := pToolLife^.time_used;

			RRes.RESULT := ADS_RDWRT_IND_NO_ERROR;

